C01829=1187.154,242.876,-63.394,-177.309,7.032,148.525
C01830=1187.149,243.125,-63.420,-177.307,7.034,148.524
C01831=1187.146,243.373,-63.446,-177.304,7.037,148.524
C01832=1187.141,243.622,-63.473,-177.302,7.039,148.524
C01833=1187.137,243.871,-63.499,-177.299,7.042,148.524
C01834=1187.132,244.119,-63.526,-177.296,7.044,148.524
C01835=1187.128,244.368,-63.552,-177.293,7.046,148.524
C01836=1187.123,244.616,-63.579,-177.291,7.048,148.523
C01837=1187.119,244.865,-63.605,-177.288,7.050,148.523
C01838=1187.114,245.114,-63.632,-177.286,7.053,148.523
C01839=1187.110,245.361,-63.658,-177.284,7.055,148.523
C01840=1187.105,245.610,-63.684,-177.280,7.058,148.523
C01841=1187.101,245.859,-63.711,-177.278,7.060,148.523
C01842=1187.096,246.107,-63.738,-177.275,7.063,148.522
C01843=1187.091,246.355,-63.765,-177.273,7.065,148.522
C01844=1187.087,246.604,-63.791,-177.270,7.068,148.522
C01845=1187.083,246.853,-63.818,-177.267,7.070,148.522
C01846=1187.079,247.101,-63.844,-177.265,7.073,148.522
C01847=1187.074,247.349,-63.871,-177.262,7.075,148.521
C01848=1187.070,247.599,-63.898,-177.260,7.077,148.521
C01849=1187.066,247.847,-63.924,-177.257,7.080,148.521
C01850=1187.061,248.096,-63.952,-177.255,7.082,148.521
C01851=1187.056,248.344,-63.979,-177.252,7.085,148.521
C01852=1187.053,248.593,-64.005,-177.250,7.087,148.521
C01853=1187.048,248.842,-64.031,-177.246,7.089,148.521
C01854=1187.043,249.090,-64.058,-177.244,7.092,148.520
C01855=1187.039,249.338,-64.085,-177.241,7.094,148.520
C01856=1187.034,249.587,-64.112,-177.239,7.096,148.520
C01857=1187.030,249.835,-64.139,-177.236,7.099,148.520
C01858=1187.026,250.084,-64.165,-177.234,7.101,148.520
C01859=1187.021,250.332,-64.193,-177.231,7.104,148.520
C01860=1187.016,250.581,-64.220,-177.229,7.106,148.520
C01861=1187.012,250.829,-64.247,-177.225,7.109,148.519
C01862=1187.008,251.078,-64.272,-177.223,7.111,148.519
C01863=1187.003,251.326,-64.299,-177.221,7.114,148.519
C01864=1186.999,251.576,-64.327,-177.218,7.116,148.519
C01865=1186.994,251.824,-64.354,-177.215,7.119,148.519
C01866=1186.990,252.072,-64.380,-177.213,7.121,148.519
C01867=1186.986,252.321,-64.408,-177.210,7.124,148.518
C01868=1186.981,252.569,-64.435,-177.208,7.126,148.518
C01869=1186.976,252.818,-64.462,-177.205,7.129,148.518
C01870=1186.972,253.066,-64.488,-177.202,7.131,148.518
C01871=1186.968,253.314,-64.516,-177.200,7.134,148.518
C01872=1186.964,253.563,-64.543,-177.197,7.136,148.518
C01873=1186.959,253.812,-64.570,-177.194,7.139,148.517
C01874=1186.955,254.060,-64.597,-177.192,7.141,148.517
C01875=1186.950,254.309,-64.624,-177.189,7.144,148.517
C01876=1186.946,254.557,-64.651,-177.187,7.146,148.517
C01877=1186.941,254.805,-64.678,-177.184,7.149,148.517
C01878=1186.937,255.054,-64.705,-177.182,7.151,148.517
C01879=1186.933,255.303,-64.733,-177.179,7.153,148.517
C01880=1186.928,255.551,-64.760,-177.176,7.155,148.517
C01881=1186.924,255.799,-64.787,-177.174,7.158,148.516
C01882=1186.919,256.048,-64.814,-177.171,7.160,148.516
C01883=1186.914,256.296,-64.841,-177.168,7.163,148.516
C01884=1186.910,256.545,-64.869,-177.166,7.165,148.516
C01885=1186.907,256.793,-64.896,-177.163,7.168,148.516
C01886=1186.902,257.042,-64.923,-177.161,7.170,148.516
C01887=1186.897,257.290,-64.950,-177.158,7.173,148.516
C01888=1186.893,257.539,-64.977,-177.155,7.176,148.516
C01889=1186.889,257.787,-65.005,-177.153,7.178,148.515
C01890=1186.884,258.036,-65.032,-177.150,7.181,148.515
C01891=1186.880,258.284,-65.060,-177.148,7.183,148.515
C01892=1186.875,258.532,-65.087,-177.145,7.186,148.515
C01893=1186.871,258.781,-65.115,-177.142,7.188,148.515
C01894=1186.867,259.030,-65.142,-177.140,7.191,148.515
C01895=1186.862,259.278,-65.170,-177.138,7.193,148.515
C01896=1186.858,259.526,-65.197,-177.134,7.196,148.514
C01897=1186.854,259.775,-65.224,-177.132,7.198,148.514
C01898=1186.849,260.023,-65.252,-177.129,7.201,148.514
C01899=1186.845,260.272,-65.279,-177.127,7.204,148.514
C01900=1186.840,260.519,-65.307,-177.124,7.206,148.514
C01901=1186.836,260.769,-65.334,-177.121,7.209,148.514
C01902=1186.831,261.017,-65.361,-177.119,7.211,148.514
C01903=1186.827,261.265,-65.389,-177.116,7.214,148.514
C01904=1186.823,261.514,-65.416,-177.114,7.216,148.513
C01905=1186.818,261.762,-65.445,-177.111,7.219,148.513
C01906=1186.813,262.011,-65.472,-177.109,7.221,148.513
C01907=1186.809,262.284,-65.502,-177.106,7.224,148.513
C01908=1186.804,262.557,-65.532,-177.103,7.227,148.513
C01909=1186.799,262.830,-65.563,-177.100,7.230,148.513
C01910=1186.794,263.103,-65.593,-177.097,7.232,148.513
C01911=1186.790,263.350,-65.621,-177.094,7.235,148.513
C01912=1186.786,263.600,-65.648,-177.092,7.237,148.512
C01913=1186.781,263.847,-65.676,-177.089,7.240,148.512
C01914=1186.777,264.097,-65.704,-177.087,7.243,148.512
C01915=1186.772,264.345,-65.732,-177.084,7.245,148.512
C01916=1186.768,264.593,-65.760,-177.081,7.248,148.512
C01917=1186.764,264.842,-65.787,-177.079,7.250,148.512
C01918=1186.760,265.090,-65.815,-177.077,7.253,148.512
C01919=1186.755,265.338,-65.843,-177.074,7.255,148.512
C01920=1186.750,265.587,-65.871,-177.071,7.258,148.511
C01921=1186.746,265.835,-65.899,-177.068,7.261,148.511
C01922=1186.742,266.083,-65.926,-177.066,7.263,148.511
C01923=1186.738,266.332,-65.954,-177.064,7.266,148.511
C01924=1186.733,266.580,-65.981,-177.061,7.268,148.511
C01925=1186.729,266.829,-66.010,-177.058,7.271,148.511
C01926=1186.724,267.077,-66.038,-177.055,7.274,148.511
C01927=1186.720,267.325,-66.065,-177.053,7.276,148.511
C01928=1186.715,267.574,-66.094,-177.051,7.279,148.511
C01929=1186.711,267.822,-66.122,-177.048,7.281,148.511
C01930=1186.707,268.071,-66.150,-177.045,7.284,148.510
C01931=1186.703,268.319,-66.177,-177.042,7.287,148.510
C01932=1186.698,268.568,-66.206,-177.040,7.289,148.510
C01933=1186.694,268.816,-66.233,-177.038,7.292,148.510
C01934=1186.689,269.064,-66.261,-177.035,7.295,148.510
C01935=1186.685,269.313,-66.290,-177.032,7.297,148.510
C01936=1186.681,269.560,-66.318,-177.030,7.300,148.510
C01937=1186.676,269.810,-66.345,-177.027,7.302,148.510
C01938=1186.671,270.058,-66.373,-177.025,7.305,148.510
C01939=1186.668,270.306,-66.402,-177.022,7.308,148.510
C01940=1186.663,270.554,-66.429,-177.020,7.310,148.510
C01941=1186.659,270.803,-66.458,-177.017,7.313,148.509
C01942=1186.654,271.051,-66.486,-177.014,7.315,148.509
C01943=1186.650,271.300,-66.515,-177.012,7.318,148.509
C01944=1186.646,271.548,-66.542,-177.009,7.321,148.509
C01945=1186.642,271.796,-66.570,-177.007,7.323,148.509
C01946=1186.637,272.045,-66.599,-177.004,7.326,148.509
C01947=1186.633,272.293,-66.627,-177.001,7.329,148.509
C01948=1186.628,272.541,-66.655,-176.999,7.331,148.509
C01949=1186.624,272.790,-66.684,-176.996,7.334,148.509
C01950=1186.619,273.038,-66.712,-176.993,7.337,148.509
C01951=1186.615,273.287,-66.740,-176.991,7.339,148.509
C01952=1186.610,273.535,-66.768,-176.988,7.342,148.509
C01953=1186.607,273.783,-66.797,-176.986,7.345,148.508
C01954=1186.601,274.032,-66.825,-176.984,7.347,148.508
C01955=1186.598,274.280,-66.853,-176.981,7.350,148.508
C01956=1186.594,274.528,-66.882,-176.978,7.352,148.508
C01957=1186.589,274.776,-66.910,-176.975,7.355,148.508
C01958=1186.585,275.025,-66.939,-176.973,7.358,148.508
C01959=1186.580,275.273,-66.967,-176.971,7.360,148.508
C01960=1186.576,275.522,-66.996,-176.968,7.363,148.508
C01961=1186.571,275.770,-67.023,-176.965,7.366,148.508
C01962=1186.567,276.018,-67.053,-176.963,7.369,148.508
C01963=1186.564,276.267,-67.081,-176.960,7.372,148.508
C01964=1186.558,276.515,-67.109,-176.958,7.375,148.508
C01965=1186.555,276.764,-67.137,-176.955,7.376,148.507
C01966=1186.550,277.012,-67.166,-176.952,7.379,148.507
C01967=1186.545,277.260,-67.195,-176.949,7.382,148.507
C01968=1186.542,277.509,-67.223,-176.947,7.385,148.507
C01969=1186.537,277.757,-67.252,-176.945,7.388,148.507
C01970=1186.533,278.005,-67.281,-176.942,7.391,148.507
C01971=1186.529,278.254,-67.309,-176.940,7.393,148.507
C01972=1186.524,278.502,-67.338,-176.937,7.396,148.507
C01973=1186.520,278.750,-67.367,-176.934,7.399,148.507
C01974=1186.515,278.998,-67.395,-176.932,7.401,148.507
C01975=1186.511,279.246,-67.423,-176.929,7.404,148.507
C01976=1186.507,279.495,-67.453,-176.926,7.406,148.507
C01977=1186.502,279.743,-67.481,-176.923,7.409,148.507
C01978=1186.498,279.992,-67.509,-176.921,7.412,148.507
C01979=1186.494,280.240,-67.539,-176.919,7.415,148.506
C01980=1186.489,280.488,-67.567,-176.916,7.418,148.506
C01981=1186.485,280.736,-67.596,-176.914,7.420,148.506
C01982=1186.481,280.985,-67.625,-176.911,7.423,148.506
C01983=1186.477,281.233,-67.654,-176.908,7.426,148.506
C01984=1186.472,281.481,-67.682,-176.906,7.428,148.506
C01985=1186.468,281.730,-67.710,-176.903,7.431,148.506
C01986=1186.464,281.978,-67.740,-176.901,7.434,148.506
C01987=1186.459,282.226,-67.768,-176.899,7.436,148.506
C01988=1186.455,282.475,-67.798,-176.896,7.439,148.506
C01989=1186.450,282.723,-67.827,-176.893,7.442,148.506
C01990=1186.447,282.971,-67.855,-176.890,7.445,148.506
C01991=1186.442,283.219,-67.884,-176.888,7.447,148.506
C01992=1186.437,283.468,-67.913,-176.885,7.450,148.506
C01993=1186.433,283.716,-67.943,-176.883,7.453,148.506
C01994=1186.428,283.964,-67.971,-176.881,7.455,148.506
C01995=1186.425,284.212,-68.000,-176.878,7.458,148.506
C01996=1186.421,284.461,-68.029,-176.875,7.461,148.506
C01997=1186.416,284.709,-68.058,-176.872,7.464,148.506
C01998=1186.411,284.957,-68.087,-176.870,7.467,148.506
C01999=1186.407,285.205,-68.117,-176.867,7.469,148.505
C02000=1186.403,285.454,-68.145,-176.864,7.472,148.505
C02001=1186.399,285.702,-68.174,-176.862,7.474,148.505
C02002=1186.395,285.950,-68.204,-176.860,7.477,148.505
C02003=1186.390,286.199,-68.232,-176.857,7.480,148.505
C02004=1186.386,286.447,-68.261,-176.854,7.483,148.505
C02005=1186.381,286.695,-68.291,-176.852,7.486,148.505
C02006=1186.377,286.943,-68.320,-176.849,7.489,148.505
C02007=1186.373,287.192,-68.349,-176.846,7.492,148.505
C02008=1186.368,287.440,-68.378,-176.844,7.495,148.505
C02009=1186.364,287.688,-68.408,-176.842,7.497,148.505
C02010=1186.360,287.936,-68.437,-176.839,7.500,148.505
C02011=1186.355,288.211,-68.469,-176.836,7.503,148.505
C02012=1186.350,288.486,-68.501,-176.833,7.506,148.505
C02013=1186.345,288.760,-68.534,-176.831,7.509,148.505
C02014=1186.340,289.035,-68.566,-176.827,7.513,148.505
C02015=1186.336,289.283,-68.596,-176.825,7.515,148.505
C02016=1186.332,289.532,-68.625,-176.823,7.518,148.505
C02017=1186.327,289.779,-68.654,-176.820,7.521,148.505
C02018=1186.323,290.028,-68.684,-176.818,7.523,148.505
C02019=1186.319,290.276,-68.713,-176.815,7.526,148.505
C02020=1186.315,290.524,-68.743,-176.812,7.529,148.505
C02021=1186.311,290.772,-68.772,-176.810,7.532,148.504
C02022=1186.306,291.021,-68.802,-176.807,7.534,148.504
C02023=1186.302,291.269,-68.831,-176.805,7.537,148.504
C02024=1186.298,291.517,-68.860,-176.802,7.540,148.504
C02025=1186.293,291.765,-68.890,-176.800,7.543,148.505
C02026=1186.289,292.013,-68.919,-176.798,7.545,148.504
C02027=1186.285,292.261,-68.948,-176.795,7.548,148.504
C02028=1186.281,292.510,-68.978,-176.792,7.551,148.504
C02029=1186.277,292.758,-69.007,-176.789,7.554,148.504
C02030=1186.272,293.006,-69.037,-176.787,7.557,148.504
C02031=1186.268,293.254,-69.066,-176.785,7.560,148.504
C02032=1186.263,293.503,-69.096,-176.782,7.563,148.504
C02033=1186.259,293.751,-69.126,-176.779,7.566,148.504
C02034=1186.255,293.999,-69.155,-176.776,7.569,148.504
C02035=1186.251,294.248,-69.185,-176.774,7.571,148.504
C02036=1186.247,294.496,-69.214,-176.771,7.574,148.504
C02037=1186.243,294.744,-69.244,-176.769,7.577,148.504
C02038=1186.238,294.992,-69.274,-176.766,7.580,148.504
C02039=1186.234,295.240,-69.304,-176.764,7.582,148.504
C02040=1186.229,295.489,-69.333,-176.762,7.585,148.504
C02041=1186.225,295.737,-69.363,-176.759,7.588,148.504
C02042=1186.221,295.985,-69.392,-176.756,7.591,148.504
C02043=1186.217,296.233,-69.422,-176.754,7.594,148.504
C02044=1186.212,296.482,-69.452,-176.751,7.596,148.504
C02045=1186.208,296.730,-69.482,-176.749,7.599,148.504
C02046=1186.204,296.978,-69.511,-176.746,7.602,148.504
C02047=1186.200,297.226,-69.541,-176.743,7.605,148.504
C02048=1186.195,297.474,-69.572,-176.741,7.608,148.504
C02049=1186.191,297.723,-69.601,-176.739,7.611,148.504
C02050=1186.187,297.970,-69.631,-176.736,7.614,148.504
C02051=1186.182,298.219,-69.661,-176.733,7.617,148.504
C02052=1186.178,298.467,-69.691,-176.731,7.620,148.504
C02053=1186.174,298.715,-69.721,-176.728,7.622,148.504
C02054=1186.170,298.963,-69.750,-176.726,7.625,148.504
C02055=1186.165,299.212,-69.780,-176.723,7.628,148.504
C02056=1186.161,299.459,-69.810,-176.720,7.631,148.504
C02057=1186.157,299.707,-69.840,-176.718,7.634,148.504
C02058=1186.152,299.955,-69.871,-176.716,7.637,148.504
C02059=1186.148,300.204,-69.900,-176.713,7.640,148.504
C02060=1186.144,300.451,-69.930,-176.711,7.643,148.504
C02061=1186.139,300.700,-69.960,-176.708,7.646,148.504
C02062=1186.136,300.948,-69.991,-176.705,7.649,148.504
C02063=1186.131,301.197,-70.021,-176.703,7.651,148.504
C02064=1186.127,301.444,-70.051,-176.701,7.654,148.504
C02065=1186.123,301.693,-70.081,-176.698,7.657,148.504
C02066=1186.118,301.941,-70.111,-176.695,7.660,148.504
C02067=1186.114,302.189,-70.141,-176.693,7.663,148.504
C02068=1186.110,302.437,-70.172,-176.690,7.665,148.504
C02069=1186.105,302.685,-70.201,-176.688,7.668,148.504
C02070=1186.101,302.933,-70.232,-176.685,7.672,148.504
C02071=1186.097,303.182,-70.262,-176.683,7.675,148.504
C02072=1186.093,303.430,-70.292,-176.680,7.678,148.504
C02073=1186.089,303.678,-70.323,-176.678,7.680,148.504
C02074=1186.085,303.926,-70.352,-176.675,7.683,148.504
C02075=1186.080,304.174,-70.383,-176.672,7.686,148.504
C02076=1186.076,304.422,-70.412,-176.670,7.689,148.504
C02077=1186.071,304.670,-70.443,-176.667,7.692,148.504
C02078=1186.067,304.919,-70.474,-176.665,7.695,148.504
C02079=1186.063,305.166,-70.504,-176.663,7.697,148.504
C02080=1186.058,305.415,-70.534,-176.660,7.700,148.504
C02081=1186.055,305.663,-70.564,-176.658,7.704,148.504
C02082=1186.050,305.911,-70.595,-176.655,7.707,148.504
C02083=1186.046,306.159,-70.625,-176.652,7.710,148.504
C02084=1186.042,306.408,-70.656,-176.649,7.713,148.504
C02085=1186.038,306.655,-70.686,-176.647,7.715,148.504
C02086=1186.033,306.903,-70.717,-176.645,7.718,148.504
C02087=1186.029,307.151,-70.748,-176.642,7.721,148.504
C02088=1186.024,307.399,-70.777,-176.640,7.724,148.504
C02089=1186.020,307.648,-70.808,-176.637,7.727,148.504
C02090=1186.017,307.896,-70.838,-176.635,7.730,148.504
C02091=1186.012,308.144,-70.869,-176.633,7.733,148.504
C02092=1186.007,308.392,-70.900,-176.630,7.736,148.504
C02093=1186.004,308.640,-70.930,-176.627,7.739,148.504
C02094=1185.999,308.889,-70.960,-176.625,7.742,148.505
C02095=1185.994,309.137,-70.991,-176.622,7.745,148.505
C02096=1185.991,309.384,-71.021,-176.619,7.748,148.505
C02097=1185.987,309.633,-71.052,-176.617,7.750,148.504
C02098=1185.982,309.881,-71.083,-176.615,7.753,148.505
C02099=1185.978,310.128,-71.113,-176.612,7.756,148.505
C02100=1185.974,310.376,-71.144,-176.610,7.759,148.505
C02101=1185.969,310.625,-71.175,-176.607,7.762,148.505
C02102=1185.966,310.873,-71.205,-176.605,7.766,148.505
C02103=1185.961,311.121,-71.236,-176.602,7.768,148.505
C02104=1185.957,311.369,-71.267,-176.600,7.771,148.505
C02105=1185.952,311.617,-71.298,-176.598,7.774,148.505
C02106=1185.949,311.865,-71.328,-176.595,7.777,148.505
C02107=1185.944,312.113,-71.359,-176.592,7.780,148.505
C02108=1185.940,312.362,-71.390,-176.589,7.783,148.505
C02109=1185.935,312.609,-71.421,-176.587,7.786,148.505
C02110=1185.931,312.857,-71.451,-176.585,7.789,148.505
C02111=1185.928,313.105,-71.483,-176.582,7.792,148.505
C02112=1185.923,313.353,-71.514,-176.580,7.795,148.505
C02113=1185.918,313.601,-71.544,-176.577,7.798,148.505
C02114=1185.914,313.850,-71.576,-176.575,7.801,148.505
C02115=1185.910,314.126,-71.610,-176.572,7.804,148.505
C02116=1185.905,314.403,-71.644,-176.570,7.807,148.505
C02117=1185.900,314.679,-71.679,-176.566,7.811,148.505
C02118=1185.895,314.955,-71.713,-176.564,7.814,148.505
C02119=1185.891,315.204,-71.744,-176.561,7.817,148.506
C02120=1185.887,315.452,-71.775,-176.559,7.820,148.506
C02121=1185.884,315.700,-71.806,-176.556,7.823,148.506
C02122=1185.879,315.948,-71.837,-176.554,7.827,148.506
C02123=1185.875,316.196,-71.868,-176.552,7.829,148.506
C02124=1185.871,316.444,-71.899,-176.549,7.832,148.506
C02125=1185.866,316.692,-71.930,-176.547,7.835,148.506
C02126=1185.862,316.940,-71.962,-176.544,7.838,148.506
C02127=1185.858,317.188,-71.992,-176.541,7.841,148.506
C02128=1185.853,317.436,-72.023,-176.539,7.845,148.506
C02129=1185.849,317.684,-72.055,-176.536,7.848,148.506
C02130=1185.845,317.932,-72.086,-176.534,7.850,148.506
C02131=1185.841,318.181,-72.117,-176.532,7.853,148.506
C02132=1185.837,318.428,-72.148,-176.529,7.856,148.506
C02133=1185.833,318.676,-72.179,-176.527,7.859,148.506
C02134=1185.829,318.924,-72.210,-176.524,7.862,148.506
C02135=1185.825,319.172,-72.242,-176.521,7.865,148.506
C02136=1185.821,319.420,-72.273,-176.519,7.869,148.507
C02137=1185.817,319.668,-72.304,-176.516,7.872,148.507
C02138=1185.812,319.916,-72.335,-176.514,7.875,148.507
C02139=1185.808,320.164,-72.366,-176.512,7.877,148.507
C02140=1185.804,320.412,-72.398,-176.509,7.880,148.507
C02141=1185.799,320.660,-72.429,-176.507,7.884,148.507
C02142=1185.795,320.908,-72.460,-176.504,7.887,148.507
C02143=1185.790,321.156,-72.492,-176.502,7.890,148.507
C02144=1185.787,321.404,-72.524,-176.499,7.893,148.507
C02145=1185.782,321.652,-72.555,-176.497,7.896,148.507
C02146=1185.778,321.900,-72.587,-176.494,7.899,148.507
C02147=1185.774,322.149,-72.618,-176.493,7.902,148.508
C02148=1185.770,322.396,-72.649,-176.490,7.905,148.508
C02149=1185.766,322.645,-72.680,-176.487,7.908,148.508
C02150=1185.762,322.892,-72.712,-176.485,7.911,148.508
C02151=1185.758,323.140,-72.744,-176.482,7.914,148.508
C02152=1185.753,323.388,-72.775,-176.480,7.917,148.508
C02153=1185.750,323.636,-72.806,-176.477,7.920,148.508
C02154=1185.745,323.884,-72.838,-176.475,7.924,148.508
C02155=1185.741,324.132,-72.870,-176.472,7.927,148.508
C02156=1185.736,324.380,-72.901,-176.470,7.930,148.508
C02157=1185.732,324.628,-72.933,-176.468,7.932,148.508
C02158=1185.729,324.876,-72.965,-176.466,7.935,148.509
C02159=1185.724,325.124,-72.996,-176.463,7.938,148.509
C02160=1185.720,325.372,-73.027,-176.461,7.942,148.509
C02161=1185.715,325.619,-73.059,-176.458,7.945,148.509
C02162=1185.712,325.868,-73.091,-176.456,7.948,148.509
C02163=1185.708,326.116,-73.122,-176.453,7.951,148.509
C02164=1185.703,326.364,-73.154,-176.451,7.954,148.509
C02165=1185.699,326.612,-73.186,-176.448,7.957,148.509
C02166=1185.695,326.859,-73.218,-176.446,7.961,148.509
C02167=1185.691,327.107,-73.250,-176.444,7.963,148.509
C02168=1185.687,327.355,-73.282,-176.442,7.966,148.509
C02169=1185.682,327.604,-73.313,-176.439,7.969,148.509
C02170=1185.678,327.852,-73.345,-176.437,7.973,148.510
C02171=1185.674,328.099,-73.376,-176.434,7.976,148.510
C02172=1185.670,328.347,-73.408,-176.432,7.979,148.510
C02173=1185.666,328.595,-73.441,-176.429,7.982,148.510
C02174=1185.661,328.843,-73.472,-176.427,7.985,148.510
C02175=1185.658,329.091,-73.504,-176.424,7.989,148.510
C02176=1185.653,329.339,-73.536,-176.422,7.992,148.510
C02177=1185.649,329.586,-73.568,-176.419,7.995,148.511
C02178=1185.645,329.834,-73.600,-176.418,7.997,148.511
C02179=1185.641,330.083,-73.632,-176.415,8.000,148.511
C02180=1185.636,330.330,-73.664,-176.413,8.004,148.511
C02181=1185.633,330.578,-73.695,-176.410,8.007,148.511
C02182=1185.628,330.827,-73.728,-176.408,8.010,148.511
C02183=1185.624,331.074,-73.759,-176.406,8.013,148.511
C02184=1185.620,331.322,-73.792,-176.403,8.016,148.511
C02185=1185.616,331.570,-73.824,-176.401,8.020,148.512
C02186=1185.612,331.818,-73.855,-176.398,8.023,148.512
C02187=1185.607,332.066,-73.887,-176.396,8.026,148.512
C02188=1185.603,332.314,-73.919,-176.393,8.029,148.512
C02189=1185.599,332.562,-73.952,-176.391,8.032,148.512
C02190=1185.595,332.809,-73.984,-176.389,8.035,148.512
C02191=1185.591,333.057,-74.016,-176.387,8.038,148.512
C02192=1185.587,333.305,-74.048,-176.384,8.041,148.512
C02193=1185.583,333.553,-74.080,-176.382,8.044,148.513
C02194=1185.578,333.801,-74.112,-176.380,8.048,148.513
C02195=1185.574,334.049,-74.144,-176.377,8.051,148.513
C02196=1185.570,334.297,-74.177,-176.375,8.054,148.513
C02197=1185.567,334.545,-74.209,-176.372,8.057,148.513
C02198=1185.561,334.793,-74.241,-176.370,8.061,148.513
C02199=1185.558,335.041,-74.273,-176.367,8.064,148.513
C02200=1185.554,335.288,-74.306,-176.365,8.067,148.514
C02201=1185.550,335.536,-74.338,-176.363,8.070,148.514
C02202=1185.545,335.785,-74.370,-176.360,8.073,148.514
C02203=1185.541,336.032,-74.403,-176.358,8.077,148.514
C02204=1185.537,336.280,-74.435,-176.356,8.079,148.514
C02205=1185.533,336.528,-74.467,-176.354,8.083,148.514
C02206=1185.529,336.776,-74.500,-176.351,8.086,148.514
C02207=1185.525,337.024,-74.532,-176.349,8.089,148.515
C02208=1185.520,337.271,-74.564,-176.347,8.092,148.515
C02209=1185.516,337.519,-74.597,-176.344,8.095,148.515
C02210=1185.512,337.767,-74.630,-176.342,8.098,148.515
C02211=1185.508,338.015,-74.662,-176.340,8.102,148.515
C02212=1185.504,338.263,-74.695,-176.337,8.105,148.515
C02213=1185.500,338.510,-74.726,-176.335,8.108,148.516
C02214=1185.496,338.758,-74.759,-176.333,8.112,148.516
C02215=1185.491,339.006,-74.792,-176.330,8.115,148.516
C02216=1185.488,339.254,-74.824,-176.328,8.118,148.516
C02217=1185.483,339.502,-74.857,-176.326,8.121,148.516
C02218=1185.479,339.750,-74.890,-176.323,8.125,148.517
C02219=1185.475,340.029,-74.926,-176.321,8.128,148.517
C02220=1185.470,340.308,-74.962,-176.318,8.131,148.517
C02221=1185.465,340.587,-74.999,-176.316,8.135,148.517
C02222=1185.460,340.865,-75.036,-176.313,8.139,148.517
C02223=1185.456,341.113,-75.069,-176.311,8.142,148.518
C02224=1185.452,341.361,-75.101,-176.309,8.145,148.518
C02225=1185.448,341.609,-75.134,-176.307,8.148,148.518
C02226=1185.444,341.857,-75.167,-176.304,8.152,148.518
C02227=1185.440,342.105,-75.200,-176.302,8.155,148.518
C02228=1185.436,342.352,-75.232,-176.299,8.158,148.518
C02229=1185.432,342.601,-75.265,-176.297,8.161,148.519
C02230=1185.428,342.848,-75.298,-176.295,8.165,148.519
C02231=1185.423,343.095,-75.331,-176.293,8.168,148.519
C02232=1185.419,343.343,-75.362,-176.290,8.171,148.519
C02233=1185.415,343.591,-75.396,-176.288,8.175,148.519
C02234=1185.411,343.839,-75.429,-176.286,8.178,148.520
C02235=1185.407,344.087,-75.461,-176.284,8.181,148.520
C02236=1185.402,344.335,-75.494,-176.281,8.185,148.520
C02237=1185.398,344.583,-75.528,-176.279,8.188,148.520
C02238=1185.395,344.830,-75.560,-176.277,8.191,148.521
C02239=1185.390,345.078,-75.593,-176.275,8.195,148.521
C02240=1185.386,345.326,-75.626,-176.273,8.197,148.521
C02241=1185.382,345.574,-75.659,-176.271,8.200,148.521
C02242=1185.378,345.822,-75.692,-176.268,8.204,148.521
C02243=1185.374,346.069,-75.725,-176.266,8.207,148.522
C02244=1185.370,346.317,-75.758,-176.264,8.210,148.522
C02245=1185.366,346.565,-75.790,-176.262,8.214,148.522
C02246=1185.362,346.813,-75.823,-176.259,8.217,148.522
C02247=1185.358,347.060,-75.856,-176.257,8.220,148.522
C02248=1185.354,347.308,-75.890,-176.255,8.224,148.523
C02249=1185.349,347.556,-75.923,-176.253,8.227,148.523
C02250=1185.345,347.804,-75.956,-176.250,8.230,148.523
C02251=1185.341,348.051,-75.989,-176.248,8.234,148.523
C02252=1185.337,348.299,-76.022,-176.246,8.237,148.524
C02253=1185.333,348.547,-76.055,-176.244,8.240,148.524
C02254=1185.329,348.795,-76.089,-176.241,8.244,148.524
C02255=1185.325,349.042,-76.122,-176.239,8.247,148.524
C02256=1185.321,349.290,-76.155,-176.237,8.250,148.524
C02257=1185.316,349.538,-76.188,-176.235,8.254,148.525
C02258=1185.312,349.785,-76.221,-176.233,8.257,148.525
C02259=1185.308,350.033,-76.254,-176.230,8.260,148.525
C02260=1185.304,350.281,-76.287,-176.228,8.264,148.526
C02261=1185.300,350.529,-76.321,-176.226,8.267,148.526
C02262=1185.296,350.776,-76.354,-176.224,8.270,148.526
C02263=1185.292,351.025,-76.387,-176.221,8.274,148.526
C02264=1185.288,351.273,-76.420,-176.220,8.277,148.527
C02265=1185.284,351.520,-76.454,-176.217,8.281,148.527
C02266=1185.280,351.768,-76.487,-176.215,8.284,148.527
C02267=1185.276,352.016,-76.520,-176.213,8.287,148.527
C02268=1185.272,352.263,-76.554,-176.211,8.291,148.528
C02269=1185.268,352.511,-76.587,-176.209,8.294,148.528
C02270=1185.263,352.758,-76.620,-176.207,8.297,148.528
C02271=1185.259,353.006,-76.654,-176.205,8.300,148.528
C02272=1185.254,353.254,-76.687,-176.203,8.303,148.529
C02273=1185.251,353.503,-76.721,-176.201,8.307,148.529
C02274=1185.247,353.750,-76.754,-176.199,8.310,148.529
C02275=1185.243,353.997,-76.788,-176.196,8.314,148.529
C02276=1185.239,354.245,-76.821,-176.194,8.317,148.530
C02277=1185.235,354.493,-76.854,-176.192,8.321,148.530
C02278=1185.231,354.740,-76.888,-176.190,8.324,148.530
C02279=1185.226,354.988,-76.922,-176.188,8.327,148.531
C02280=1185.222,355.236,-76.955,-176.186,8.331,148.531
C02281=1185.219,355.484,-76.989,-176.184,8.334,148.531
C02282=1185.214,355.731,-77.022,-176.181,8.337,148.531
C02283=1185.210,355.979,-77.055,-176.180,8.341,148.532
C02284=1185.207,356.226,-77.089,-176.177,8.344,148.532
C02285=1185.202,356.475,-77.123,-176.176,8.348,148.532
C02286=1185.198,356.723,-77.156,-176.173,8.351,148.533
C02287=1185.194,356.970,-77.190,-176.171,8.355,148.533
C02288=1185.190,357.217,-77.223,-176.169,8.358,148.533
C02289=1185.186,357.465,-77.258,-176.167,8.362,148.534
C02290=1185.182,357.713,-77.291,-176.165,8.365,148.534
C02291=1185.178,357.961,-77.325,-176.163,8.369,148.534
C02292=1185.174,358.208,-77.358,-176.161,8.372,148.534
C02293=1185.169,358.456,-77.392,-176.159,8.376,148.535
C02294=1185.165,358.703,-77.426,-176.157,8.379,148.535
C02295=1185.162,358.952,-77.460,-176.155,8.382,148.536
C02296=1185.158,359.199,-77.493,-176.152,8.386,148.536
C02297=1185.153,359.447,-77.527,-176.151,8.389,148.536
C02298=1185.149,359.694,-77.561,-176.148,8.393,148.536
C02299=1185.146,359.942,-77.595,-176.147,8.396,148.537
C02300=1185.141,360.190,-77.629,-176.145,8.400,148.537
C02301=1185.137,360.437,-77.663,-176.143,8.403,148.538
C02302=1185.134,360.685,-77.696,-176.141,8.407,148.538
C02303=1185.129,360.933,-77.731,-176.139,8.409,148.538
C02304=1185.125,361.180,-77.764,-176.137,8.413,148.539
C02305=1185.121,361.428,-77.798,-176.135,8.417,148.539
C02306=1185.117,361.676,-77.833,-176.133,8.420,148.539
C02307=1185.113,361.923,-77.866,-176.131,8.424,148.540
C02308=1185.109,362.171,-77.900,-176.130,8.427,148.540
C02309=1185.105,362.419,-77.934,-176.127,8.431,148.540
C02310=1185.101,362.666,-77.968,-176.126,8.434,148.541
C02311=1185.097,362.914,-78.002,-176.124,8.438,148.541
C02312=1185.093,363.162,-78.036,-176.122,8.441,148.542
C02313=1185.089,363.409,-78.070,-176.120,8.444,148.542
C02314=1185.085,363.657,-78.104,-176.118,8.448,148.542
C02315=1185.081,363.905,-78.138,-176.117,8.451,148.543
C02316=1185.077,364.153,-78.172,-176.115,8.455,148.543
C02317=1185.073,364.400,-78.206,-176.113,8.458,148.544
C02318=1185.069,364.648,-78.241,-176.111,8.462,148.544
C02319=1185.065,364.895,-78.275,-176.109,8.465,148.544
C02320=1185.061,365.142,-78.309,-176.108,8.468,148.545
C02321=1185.057,365.391,-78.343,-176.106,8.472,148.545
C02322=1185.053,365.638,-78.377,-176.104,8.475,148.545
C02323=1185.048,365.920,-78.416,-176.102,8.479,148.546
C02324=1185.044,366.201,-78.455,-176.100,8.483,148.546
C02325=1185.039,366.481,-78.493,-176.098,8.487,148.547
C02326=1185.034,366.763,-78.533,-176.097,8.491,148.547
C02327=1185.031,367.012,-78.566,-176.095,8.495,148.548
C02328=1185.026,367.259,-78.601,-176.093,8.498,148.548
C02329=1185.022,367.506,-78.635,-176.092,8.501,148.549
C02330=1185.018,367.754,-78.669,-176.090,8.505,148.549
C02331=1185.014,368.002,-78.704,-176.088,8.508,148.550
C02332=1185.010,368.249,-78.738,-176.086,8.512,148.550
C02333=1185.006,368.497,-78.773,-176.085,8.515,148.550
C02334=1185.002,368.744,-78.807,-176.083,8.518,148.551
C02335=1184.998,368.992,-78.841,-176.081,8.522,148.551
C02336=1184.994,369.239,-78.875,-176.080,8.526,148.552
C02337=1184.991,369.487,-78.910,-176.079,8.529,148.552
C02338=1184.986,369.735,-78.945,-176.077,8.532,148.553
C02339=1184.982,369.982,-78.978,-176.075,8.536,148.553
C02340=1184.978,370.230,-79.013,-176.074,8.539,148.553
C02341=1184.974,370.477,-79.047,-176.072,8.542,148.554
C02342=1184.970,370.725,-79.082,-176.071,8.546,148.555
C02343=1184.966,370.973,-79.116,-176.070,8.549,148.555
C02344=1184.963,371.220,-79.151,-176.068,8.553,148.555
C02345=1184.958,371.468,-79.185,-176.066,8.557,148.556
C02346=1184.954,371.716,-79.220,-176.065,8.559,148.556
C02347=1184.950,371.963,-79.254,-176.063,8.563,148.557
C02348=1184.946,372.210,-79.288,-176.063,8.566,148.557
C02349=1184.942,372.458,-79.324,-176.061,8.570,148.558
C02350=1184.938,372.705,-79.358,-176.059,8.573,148.558
C02351=1184.934,372.953,-79.393,-176.058,8.576,148.559
C02352=1184.930,373.201,-79.427,-176.056,8.580,148.559
C02353=1184.926,373.448,-79.461,-176.055,8.583,148.560
C02354=1184.922,373.696,-79.496,-176.054,8.587,148.560
C02355=1184.918,373.943,-79.531,-176.052,8.590,148.561
C02356=1184.914,374.191,-79.566,-176.051,8.594,148.561
C02357=1184.910,374.439,-79.600,-176.050,8.596,148.562
C02358=1184.906,374.686,-79.634,-176.048,8.600,148.562
C02359=1184.902,374.934,-79.669,-176.047,8.603,148.563
C02360=1184.897,375.181,-79.704,-176.046,8.607,148.563
C02361=1184.894,375.429,-79.739,-176.045,8.610,148.564
C02362=1184.890,375.676,-79.773,-176.043,8.614,148.564
C02363=1184.886,375.924,-79.808,-176.042,8.617,148.565
C02364=1184.881,376.171,-79.843,-176.041,8.620,148.565
C02365=1184.878,376.419,-79.877,-176.040,8.623,148.566
C02366=1184.874,376.667,-79.912,-176.039,8.627,148.567
C02367=1184.870,376.914,-79.947,-176.037,8.630,148.567
C02368=1184.866,377.162,-79.982,-176.036,8.633,148.568
C02369=1184.861,377.409,-80.017,-176.035,8.636,148.568
C02370=1184.859,377.657,-80.052,-176.034,8.640,148.569
C02371=1184.854,377.904,-80.086,-176.033,8.643,148.569
C02372=1184.850,378.152,-80.121,-176.032,8.646,148.570
C02373=1184.846,378.399,-80.156,-176.030,8.650,148.570
C02374=1184.842,378.647,-80.191,-176.029,8.653,148.571
C02375=1184.837,378.894,-80.225,-176.029,8.656,148.571
C02376=1184.834,379.142,-80.260,-176.027,8.660,148.572
C02377=1184.830,379.390,-80.295,-176.026,8.663,148.572
C02378=1184.826,379.637,-80.330,-176.025,8.666,148.573
C02379=1184.822,379.885,-80.365,-176.024,8.669,148.574
C02380=1184.817,380.132,-80.400,-176.023,8.673,148.574
C02381=1184.814,380.380,-80.435,-176.022,8.676,148.575
C02382=1184.809,380.627,-80.470,-176.021,8.679,148.575
C02383=1184.806,380.874,-80.505,-176.021,8.682,148.576
C02384=1184.802,381.122,-80.539,-176.019,8.685,148.576
C02385=1184.798,381.369,-80.575,-176.018,8.689,148.577
C02386=1184.794,381.617,-80.609,-176.017,8.692,148.578
C02387=1184.790,381.864,-80.645,-176.016,8.695,148.578
C02388=1184.786,382.112,-80.680,-176.015,8.698,148.579
C02389=1184.782,382.360,-80.715,-176.015,8.701,148.579
C02390=1184.778,382.607,-80.750,-176.014,8.704,148.580
C02391=1184.774,382.855,-80.785,-176.013,8.707,148.580
C02392=1184.769,383.102,-80.820,-176.012,8.711,148.581
C02393=1184.766,383.349,-80.855,-176.011,8.714,148.582
C02394=1184.762,383.598,-80.890,-176.011,8.717,148.582
C02395=1184.758,383.844,-80.925,-176.010,8.720,148.583
C02396=1184.754,384.093,-80.960,-176.009,8.723,148.583
C02397=1184.751,384.340,-80.995,-176.008,8.726,148.584
C02398=1184.746,384.586,-81.030,-176.007,8.729,148.585
C02399=1184.742,384.835,-81.065,-176.007,8.733,148.585
C02400=1184.739,385.082,-81.100,-176.006,8.736,148.586
C02401=1184.734,385.330,-81.135,-176.005,8.739,148.587
C02402=1184.731,385.577,-81.170,-176.005,8.742,148.587
C02403=1184.726,385.824,-81.206,-176.004,8.745,148.588
C02404=1184.722,386.072,-81.240,-176.003,8.747,148.588
C02405=1184.719,386.319,-81.276,-176.003,8.750,148.589
C02406=1184.714,386.567,-81.310,-176.002,8.754,148.590
C02407=1184.710,386.814,-81.346,-176.001,8.757,148.590
C02408=1184.707,387.062,-81.382,-176.001,8.760,148.591
C02409=1184.702,387.309,-81.416,-176.000,8.762,148.591
C02410=1184.699,387.557,-81.452,-176.000,8.765,148.592
C02411=1184.695,387.804,-81.487,-175.999,8.769,148.593
C02412=1184.690,388.052,-81.522,-175.998,8.772,148.593
C02413=1184.687,388.299,-81.557,-175.998,8.774,148.594
C02414=1184.683,388.547,-81.593,-175.997,8.777,148.594
C02415=1184.679,388.794,-81.628,-175.997,8.780,148.595
C02416=1184.674,389.042,-81.663,-175.997,8.783,148.596
C02417=1184.670,389.289,-81.699,-175.996,8.786,148.596
C02418=1184.667,389.537,-81.734,-175.996,8.789,148.597
C02419=1184.662,389.784,-81.769,-175.995,8.791,148.598
C02420=1184.658,390.032,-81.804,-175.994,8.795,148.598
C02421=1184.655,390.279,-81.840,-175.994,8.797,148.599
C02422=1184.650,390.526,-81.875,-175.994,8.800,148.599
C02423=1184.647,390.774,-81.910,-175.994,8.802,148.600
C02424=1184.643,391.022,-81.946,-175.993,8.806,148.600
C02425=1184.639,391.269,-81.981,-175.993,8.808,148.601
C02426=1184.635,391.516,-82.016,-175.992,8.811,148.602
C02427=1184.630,391.800,-82.056,-175.992,8.815,148.603
C02428=1184.626,392.084,-82.097,-175.991,8.818,148.603
C02429=1184.622,392.368,-82.138,-175.991,8.820,148.604
C02430=1184.617,392.652,-82.179,-175.991,8.824,148.605
C02431=1184.613,392.899,-82.214,-175.990,8.827,148.605
C02432=1184.608,393.147,-82.249,-175.990,8.829,148.606
C02433=1184.605,393.394,-82.284,-175.990,8.832,148.607
C02434=1184.601,393.642,-82.320,-175.989,8.835,148.607
C02435=1184.597,393.889,-82.356,-175.989,8.837,148.608
C02436=1184.593,394.136,-82.391,-175.989,8.840,148.608
C02437=1184.589,394.384,-82.426,-175.989,8.843,148.609
C02438=1184.586,394.631,-82.462,-175.988,8.845,148.610
C02439=1184.581,394.880,-82.497,-175.989,8.848,148.610
C02440=1184.577,395.126,-82.532,-175.988,8.851,148.611
C02441=1184.573,395.374,-82.568,-175.987,8.853,148.611
C02442=1184.569,395.621,-82.604,-175.988,8.856,148.612
C02443=1184.566,395.869,-82.639,-175.987,8.858,148.613
C02444=1184.561,396.116,-82.674,-175.987,8.861,148.614
C02445=1184.557,396.363,-82.710,-175.987,8.864,148.614
C02446=1184.553,396.611,-82.746,-175.987,8.866,148.615
C02447=1184.549,396.858,-82.780,-175.987,8.868,148.615
C02448=1184.545,397.106,-82.816,-175.986,8.872,148.616
C02449=1184.542,397.353,-82.852,-175.986,8.874,148.617
C02450=1184.538,397.601,-82.887,-175.986,8.876,148.617
C02451=1184.533,397.849,-82.923,-175.986,8.879,148.618
C02452=1184.529,398.095,-82.958,-175.986,8.881,148.618
C02453=1184.526,398.343,-82.994,-175.985,8.884,148.619
C02454=1184.522,398.590,-83.030,-175.986,8.886,148.620
C02455=1184.518,398.838,-83.065,-175.985,8.889,148.620
C02456=1184.513,399.085,-83.101,-175.985,8.892,148.621
C02457=1184.510,399.333,-83.136,-175.985,8.894,148.621
C02458=1184.506,399.580,-83.172,-175.984,8.896,148.622
C02459=1184.502,399.828,-83.207,-175.985,8.899,148.623
C02460=1184.498,400.074,-83.243,-175.984,8.901,148.623
C02461=1184.494,400.322,-83.279,-175.985,8.904,148.624
C02462=1184.490,400.570,-83.314,-175.984,8.906,148.624
C02463=1184.486,400.817,-83.350,-175.984,8.908,148.625
C02464=1184.483,401.065,-83.385,-175.984,8.911,148.626
C02465=1184.478,401.311,-83.421,-175.984,8.913,148.626
C02466=1184.474,401.559,-83.457,-175.984,8.916,148.627
C02467=1184.470,401.807,-83.492,-175.984,8.918,148.627
C02468=1184.467,402.054,-83.528,-175.984,8.920,148.628
C02469=1184.462,402.301,-83.563,-175.984,8.923,148.629
C02470=1184.458,402.549,-83.599,-175.984,8.925,148.629
C02471=1184.454,402.796,-83.635,-175.983,8.927,148.630
C02472=1184.451,403.044,-83.670,-175.984,8.930,148.630
C02473=1184.447,403.291,-83.706,-175.983,8.932,148.631
C02474=1184.442,403.539,-83.742,-175.983,8.935,148.632
C02475=1184.438,403.786,-83.777,-175.984,8.936,148.632
C02476=1184.435,404.034,-83.813,-175.983,8.938,148.633
C02477=1184.431,404.281,-83.848,-175.984,8.941,148.633
C02478=1184.427,404.529,-83.884,-175.983,8.943,148.634
C02479=1184.422,404.776,-83.920,-175.983,8.945,148.634
C02480=1184.419,405.023,-83.955,-175.983,8.948,148.635
C02481=1184.415,405.271,-83.991,-175.983,8.950,148.636
C02482=1184.411,405.518,-84.027,-175.983,8.952,148.636
C02483=1184.407,405.766,-84.062,-175.984,8.954,148.637
C02484=1184.403,406.013,-84.098,-175.983,8.957,148.637
C02485=1184.399,406.260,-84.133,-175.983,8.959,148.638
C02486=1184.395,406.508,-84.169,-175.983,8.961,148.639
C02487=1184.391,406.755,-84.205,-175.983,8.964,148.639
C02488=1184.388,407.002,-84.241,-175.983,8.965,148.640
C02489=1184.384,407.250,-84.277,-175.983,8.967,148.640
C02490=1184.379,407.497,-84.312,-175.983,8.970,148.641
C02491=1184.375,407.745,-84.348,-175.983,8.972,148.641
C02492=1184.372,407.992,-84.383,-175.983,8.974,148.642
C02493=1184.367,408.240,-84.420,-175.983,8.976,148.643
C02494=1184.363,408.487,-84.455,-175.983,8.978,148.643
C02495=1184.360,408.735,-84.491,-175.983,8.981,148.644
C02496=1184.356,408.982,-84.526,-175.983,8.982,148.644
C02497=1184.351,409.229,-84.563,-175.983,8.985,148.645
C02498=1184.348,409.476,-84.598,-175.983,8.987,148.645
C02499=1184.344,409.724,-84.634,-175.983,8.989,148.646
C02500=1184.340,409.972,-84.670,-175.983,8.991,148.646
C02501=1184.336,410.219,-84.706,-175.983,8.993,148.647
C02502=1184.332,410.467,-84.741,-175.983,8.995,148.648
C02503=1184.327,410.714,-84.777,-175.983,8.997,148.648
C02504=1184.324,410.961,-84.813,-175.983,8.999,148.649
C02505=1184.320,411.208,-84.849,-175.983,9.001,148.649
C02506=1184.316,411.456,-84.885,-175.984,9.003,148.650
C02507=1184.312,411.703,-84.920,-175.983,9.005,148.650
C02508=1184.309,411.951,-84.956,-175.983,9.008,148.651
C02509=1184.304,412.198,-84.992,-175.983,9.009,148.651
C02510=1184.300,412.445,-85.028,-175.983,9.011,148.652
C02511=1184.297,412.692,-85.063,-175.983,9.014,148.652
C02512=1184.292,412.940,-85.100,-175.984,9.015,148.653
C02513=1184.289,413.188,-85.135,-175.983,9.018,148.653
C02514=1184.285,413.435,-85.171,-175.984,9.019,148.654
C02515=1184.281,413.682,-85.208,-175.983,9.021,148.654
C02516=1184.277,413.929,-85.243,-175.983,9.024,148.655
C02517=1184.273,414.177,-85.278,-175.983,9.025,148.655
C02518=1184.268,414.425,-85.314,-175.984,9.028,148.656
C02519=1184.265,414.672,-85.350,-175.984,9.029,148.657
C02520=1184.261,414.919,-85.386,-175.984,9.031,148.657
C02521=1184.257,415.167,-85.422,-175.983,9.034,148.658
C02522=1184.253,415.414,-85.458,-175.984,9.035,148.658
C02523=1184.250,415.629,-85.489,-175.983,9.037,148.659
C02524=1184.246,415.844,-85.520,-175.984,9.039,148.659
C02525=1184.244,416.059,-85.551,-175.984,9.040,148.659
C02526=1184.243,416.274,-85.582,-175.983,9.042,148.660
C02527=1184.242,416.489,-85.613,-175.984,9.044,148.660
C02528=1184.242,416.703,-85.644,-175.983,9.045,148.661
C02529=1184.244,416.918,-85.675,-175.984,9.046,148.661
C02530=1184.246,417.132,-85.706,-175.983,9.048,148.662
C02531=1183.825,417.132,-85.747,-175.986,9.059,148.665
C02532=1183.822,416.917,-85.716,-175.987,9.057,148.665
C02533=1183.821,416.701,-85.685,-175.987,9.056,148.664
C02534=1183.821,416.485,-85.655,-175.987,9.054,148.664
C02535=1183.821,416.269,-85.623,-175.986,9.053,148.663
C02536=1183.822,416.052,-85.592,-175.987,9.051,148.663
C02537=1183.825,415.836,-85.561,-175.987,9.049,148.663
C02538=1183.829,415.619,-85.530,-175.986,9.048,148.662
C02539=1183.832,415.403,-85.498,-175.987,9.046,148.662
C02540=1183.836,415.155,-85.462,-175.986,9.044,148.661
C02541=1183.840,414.908,-85.426,-175.987,9.042,148.661
C02542=1183.843,414.661,-85.390,-175.987,9.040,148.660
C02543=1183.848,414.414,-85.354,-175.987,9.038,148.660
C02544=1183.852,414.166,-85.319,-175.987,9.036,148.659
C02545=1183.855,413.919,-85.283,-175.987,9.035,148.659
C02546=1183.860,413.671,-85.247,-175.986,9.032,148.658
C02547=1183.863,413.424,-85.211,-175.986,9.031,148.658
C02548=1183.867,413.176,-85.175,-175.986,9.028,148.657
C02549=1183.871,412.929,-85.139,-175.987,9.026,148.657
C02550=1183.876,412.682,-85.104,-175.986,9.025,148.656
C02551=1183.879,412.434,-85.068,-175.987,9.022,148.656
C02552=1183.883,412.187,-85.032,-175.986,9.020,148.655
C02553=1183.887,411.940,-84.996,-175.986,9.018,148.654
C02554=1183.891,411.692,-84.960,-175.986,9.016,148.654
C02555=1183.895,411.444,-84.924,-175.987,9.014,148.653
C02556=1183.899,411.197,-84.889,-175.986,9.012,148.653
C02557=1183.903,410.951,-84.853,-175.986,9.010,148.652
C02558=1183.907,410.703,-84.817,-175.986,9.008,148.652
C02559=1183.911,410.455,-84.781,-175.986,9.006,148.651
C02560=1183.914,410.208,-84.746,-175.986,9.004,148.651
C02561=1183.919,409.960,-84.709,-175.986,9.001,148.650
C02562=1183.922,409.713,-84.674,-175.986,9.000,148.649
C02563=1183.926,409.465,-84.638,-175.986,8.998,148.649
C02564=1183.931,409.219,-84.602,-175.986,8.995,148.648
C02565=1183.934,408.971,-84.566,-175.986,8.994,148.648
C02566=1183.938,408.724,-84.531,-175.986,8.991,148.647
C02567=1183.942,408.476,-84.495,-175.986,8.989,148.647
C02568=1183.946,408.228,-84.459,-175.986,8.987,148.646
C02569=1183.950,407.981,-84.424,-175.986,8.985,148.646
C02570=1183.954,407.734,-84.388,-175.986,8.983,148.645
C02571=1183.958,407.487,-84.351,-175.986,8.981,148.645
C02572=1183.962,407.239,-84.316,-175.986,8.978,148.644
C02573=1183.966,406.992,-84.280,-175.986,8.977,148.643
C02574=1183.970,406.744,-84.244,-175.986,8.974,148.643
C02575=1183.974,406.496,-84.209,-175.986,8.972,148.642
C02576=1183.978,406.250,-84.174,-175.986,8.969,148.642
C02577=1183.981,406.002,-84.138,-175.986,8.968,148.641
C02578=1183.986,405.754,-84.102,-175.986,8.966,148.641
C02579=1183.990,405.507,-84.066,-175.986,8.963,148.640
C02580=1183.993,405.259,-84.031,-175.986,8.961,148.639
C02581=1183.997,405.013,-83.996,-175.986,8.958,148.639
C02582=1184.002,404.765,-83.959,-175.986,8.956,148.638
C02583=1184.005,404.518,-83.923,-175.986,8.955,148.638
C02584=1184.009,404.270,-83.888,-175.986,8.952,148.637
C02585=1184.013,404.023,-83.851,-175.986,8.950,148.636
C02586=1184.017,403.775,-83.816,-175.986,8.948,148.636
C02587=1184.021,403.528,-83.781,-175.986,8.945,148.635
C02588=1184.025,403.281,-83.745,-175.986,8.943,148.635
C02589=1184.029,403.033,-83.709,-175.987,8.940,148.634
C02590=1184.033,402.785,-83.673,-175.986,8.938,148.633
C02591=1184.037,402.538,-83.638,-175.987,8.936,148.633
C02592=1184.041,402.291,-83.603,-175.986,8.933,148.632
C02593=1184.045,402.043,-83.567,-175.987,8.931,148.632
C02594=1184.049,401.796,-83.531,-175.987,8.929,148.631
C02595=1184.053,401.548,-83.496,-175.987,8.926,148.630
C02596=1184.056,401.301,-83.460,-175.986,8.925,148.630
C02597=1184.061,401.054,-83.425,-175.986,8.922,148.629
C02598=1184.065,400.806,-83.389,-175.987,8.920,148.629
C02599=1184.069,400.559,-83.353,-175.987,8.917,148.628
C02600=1184.072,400.311,-83.318,-175.987,8.914,148.627
C02601=1184.077,400.064,-83.282,-175.987,8.912,148.627
C02602=1184.081,399.817,-83.246,-175.987,8.909,148.626
C02603=1184.085,399.569,-83.211,-175.988,8.907,148.626
C02604=1184.088,399.322,-83.175,-175.987,8.904,148.625
C02605=1184.092,399.074,-83.140,-175.988,8.902,148.624
C02606=1184.096,398.827,-83.104,-175.988,8.900,148.624
C02607=1184.101,398.579,-83.068,-175.988,8.897,148.623
C02608=1184.104,398.332,-83.033,-175.988,8.895,148.623
C02609=1184.108,398.084,-82.997,-175.988,8.892,148.622
C02610=1184.112,397.838,-82.962,-175.988,8.890,148.621
C02611=1184.116,397.590,-82.926,-175.988,8.887,148.621
C02612=1184.120,397.342,-82.890,-175.989,8.885,148.620
C02613=1184.124,397.094,-82.855,-175.989,8.882,148.620
C02614=1184.128,396.847,-82.820,-175.989,8.880,148.619
C02615=1184.132,396.600,-82.785,-175.989,8.877,148.618
C02616=1184.136,396.352,-82.749,-175.989,8.875,148.618
C02617=1184.139,396.105,-82.714,-175.990,8.872,148.617
C02618=1184.144,395.858,-82.678,-175.989,8.869,148.616
C02619=1184.148,395.610,-82.642,-175.990,8.867,148.616
C02620=1184.152,395.363,-82.607,-175.990,8.865,148.615
C02621=1184.155,395.115,-82.571,-175.990,8.861,148.614
C02622=1184.160,394.869,-82.536,-175.991,8.859,148.614
C02623=1184.164,394.620,-82.501,-175.990,8.856,148.613
C02624=1184.167,394.373,-82.466,-175.991,8.853,148.613
C02625=1184.172,394.125,-82.430,-175.991,8.851,148.612
C02626=1184.176,393.878,-82.394,-175.991,8.848,148.611
C02627=1184.180,393.631,-82.359,-175.992,8.845,148.611
C02628=1184.183,393.383,-82.323,-175.992,8.843,148.610
C02629=1184.187,393.136,-82.288,-175.992,8.841,148.609
C02630=1184.192,392.888,-82.253,-175.993,8.837,148.609
C02631=1184.195,392.641,-82.218,-175.993,8.835,148.608
C02632=1184.200,392.358,-82.177,-175.993,8.832,148.607
C02633=1184.205,392.073,-82.136,-175.994,8.828,148.607
C02634=1184.209,391.789,-82.095,-175.994,8.825,148.606
C02635=1184.214,391.505,-82.055,-175.994,8.822,148.605
C02636=1184.217,391.258,-82.019,-175.995,8.819,148.605
C02637=1184.222,391.011,-81.984,-175.995,8.817,148.604
C02638=1184.225,390.763,-81.949,-175.996,8.814,148.603
C02639=1184.229,390.515,-81.914,-175.996,8.811,148.603
C02640=1184.233,390.268,-81.879,-175.996,8.808,148.602
C02641=1184.237,390.021,-81.843,-175.997,8.805,148.602
C02642=1184.241,389.773,-81.808,-175.997,8.803,148.601
C02643=1184.245,389.525,-81.773,-175.998,8.799,148.600
C02644=1184.249,389.278,-81.738,-175.998,8.797,148.600
C02645=1184.253,389.031,-81.702,-175.999,8.794,148.599
C02646=1184.257,388.783,-81.666,-176.000,8.791,148.599
C02647=1184.262,388.536,-81.631,-175.999,8.788,148.598
C02648=1184.265,388.288,-81.596,-176.000,8.785,148.597
C02649=1184.269,388.041,-81.560,-176.001,8.782,148.597
C02650=1184.274,387.793,-81.526,-176.001,8.779,148.596
C02651=1184.277,387.546,-81.490,-176.002,8.776,148.595
C02652=1184.281,387.298,-81.455,-176.003,8.773,148.595
C02653=1184.285,387.052,-81.420,-176.003,8.770,148.594
C02654=1184.289,386.803,-81.385,-176.003,8.768,148.593
C02655=1184.293,386.556,-81.349,-176.004,8.765,148.593
C02656=1184.297,386.309,-81.314,-176.005,8.761,148.592
C02657=1184.301,386.061,-81.279,-176.006,8.758,148.592
C02658=1184.305,385.813,-81.244,-176.006,8.755,148.591
C02659=1184.309,385.566,-81.209,-176.007,8.752,148.591
C02660=1184.313,385.319,-81.174,-176.007,8.750,148.590
C02661=1184.317,385.071,-81.138,-176.008,8.747,148.589
C02662=1184.321,384.824,-81.104,-176.009,8.743,148.589
C02663=1184.325,384.576,-81.068,-176.009,8.740,148.588
C02664=1184.328,384.329,-81.033,-176.010,8.737,148.587
C02665=1184.333,384.081,-80.998,-176.011,8.734,148.587
C02666=1184.337,383.834,-80.963,-176.012,8.731,148.586
C02667=1184.341,383.586,-80.928,-176.013,8.728,148.586
C02668=1184.345,383.339,-80.893,-176.014,8.725,148.585
C02669=1184.348,383.091,-80.858,-176.014,8.722,148.585
C02670=1184.352,382.844,-80.823,-176.015,8.719,148.584
C02671=1184.356,382.596,-80.788,-176.016,8.716,148.583
C02672=1184.360,382.349,-80.753,-176.017,8.712,148.583
C02673=1184.365,382.101,-80.718,-176.018,8.709,148.582
C02674=1184.368,381.854,-80.683,-176.018,8.706,148.582
C02675=1184.372,381.606,-80.648,-176.020,8.702,148.581
C02676=1184.377,381.359,-80.613,-176.021,8.699,148.580
C02677=1184.380,381.111,-80.578,-176.021,8.696,148.580
C02678=1184.385,380.864,-80.543,-176.022,8.693,148.579
C02679=1184.389,380.616,-80.508,-176.023,8.690,148.579
C02680=1184.393,380.369,-80.473,-176.024,8.687,148.578
C02681=1184.396,380.121,-80.438,-176.025,8.683,148.577
C02682=1184.400,379.874,-80.403,-176.027,8.680,148.577
C02683=1184.404,379.626,-80.368,-176.027,8.677,148.577
C02684=1184.408,379.379,-80.333,-176.028,8.674,148.576
C02685=1184.413,379.131,-80.298,-176.029,8.670,148.575
C02686=1184.417,378.883,-80.264,-176.030,8.667,148.575
C02687=1184.420,378.636,-80.228,-176.031,8.664,148.574
C02688=1184.425,378.388,-80.194,-176.033,8.660,148.574
C02689=1184.428,378.141,-80.159,-176.034,8.657,148.573
C02690=1184.432,377.894,-80.124,-176.035,8.654,148.573
C02691=1184.436,377.645,-80.089,-176.036,8.650,148.572
C02692=1184.441,377.399,-80.054,-176.037,8.647,148.572
C02693=1184.445,377.151,-80.019,-176.038,8.644,148.571
C02694=1184.448,376.903,-79.985,-176.039,8.640,148.570
C02695=1184.452,376.656,-79.950,-176.041,8.638,148.570
C02696=1184.457,376.409,-79.915,-176.042,8.634,148.569
C02697=1184.461,376.160,-79.881,-176.043,8.631,148.569
C02698=1184.464,375.913,-79.845,-176.044,8.628,148.568
C02699=1184.468,375.666,-79.811,-176.045,8.624,148.568
C02700=1184.472,375.418,-79.776,-176.047,8.621,148.567
C02701=1184.477,375.170,-79.742,-176.048,8.617,148.567
C02702=1184.480,374.923,-79.706,-176.049,8.614,148.566
C02703=1184.484,374.676,-79.672,-176.051,8.610,148.566
C02704=1184.488,374.428,-79.638,-176.052,8.608,148.565
C02705=1184.493,374.180,-79.603,-176.053,8.604,148.565
C02706=1184.497,373.932,-79.568,-176.055,8.601,148.564
C02707=1184.500,373.686,-79.534,-176.056,8.597,148.564
C02708=1184.504,373.437,-79.499,-176.057,8.594,148.563
C02709=1184.509,373.190,-79.464,-176.059,8.590,148.563
C02710=1184.512,372.942,-79.430,-176.060,8.587,148.562
C02711=1184.517,372.695,-79.396,-176.061,8.583,148.562
C02712=1184.520,372.447,-79.360,-176.063,8.580,148.561
C02713=1184.525,372.200,-79.326,-176.064,8.577,148.561
C02714=1184.528,371.952,-79.291,-176.066,8.573,148.560
C02715=1184.533,371.705,-79.257,-176.067,8.570,148.560
C02716=1184.537,371.457,-79.223,-176.069,8.567,148.559
C02717=1184.540,371.209,-79.188,-176.070,8.563,148.559
C02718=1184.545,370.962,-79.154,-176.071,8.560,148.558
C02719=1184.549,370.714,-79.119,-176.073,8.556,148.558
C02720=1184.553,370.467,-79.085,-176.075,8.553,148.557
C02721=1184.557,370.219,-79.050,-176.076,8.550,148.557
C02722=1184.561,369.971,-79.016,-176.078,8.546,148.556
C02723=1184.564,369.723,-78.982,-176.079,8.542,148.556
C02724=1184.569,369.476,-78.947,-176.081,8.540,148.556
C02725=1184.573,369.229,-78.913,-176.082,8.536,148.555
C02726=1184.577,368.981,-78.878,-176.084,8.532,148.555
C02727=1184.581,368.734,-78.845,-176.086,8.528,148.554
C02728=1184.585,368.485,-78.810,-176.087,8.526,148.554
C02729=1184.589,368.238,-78.775,-176.089,8.522,148.553
C02730=1184.592,367.990,-78.741,-176.090,8.518,148.553
C02731=1184.597,367.743,-78.707,-176.092,8.515,148.552
C02732=1184.601,367.496,-78.673,-176.094,8.512,148.552
C02733=1184.605,367.248,-78.638,-176.095,8.508,148.552
C02734=1184.609,367.000,-78.604,-176.097,8.505,148.551
C02735=1184.613,366.753,-78.570,-176.099,8.501,148.551
C02736=1184.617,366.472,-78.531,-176.100,8.497,148.550
C02737=1184.622,366.190,-78.491,-176.102,8.494,148.550
C02738=1184.627,365.908,-78.453,-176.105,8.489,148.549
C02739=1184.631,365.627,-78.414,-176.106,8.485,148.549
C02740=1184.635,365.379,-78.380,-176.108,8.482,148.548
C02741=1184.639,365.132,-78.345,-176.110,8.478,148.548
C02742=1184.643,364.884,-78.311,-176.111,8.475,148.547
C02743=1184.647,364.636,-78.278,-176.113,8.472,148.547
C02744=1184.651,364.388,-78.243,-176.115,8.469,148.547
C02745=1184.655,364.141,-78.209,-176.117,8.465,148.546
C02746=1184.660,363.894,-78.175,-176.119,8.461,148.546
C02747=1184.663,363.646,-78.140,-176.121,8.458,148.546
C02748=1184.667,363.398,-78.107,-176.123,8.454,148.545
C02749=1184.672,363.151,-78.073,-176.124,8.452,148.545
C02750=1184.675,362.903,-78.039,-176.126,8.448,148.544
C02751=1184.680,362.655,-78.005,-176.128,8.444,148.544
C02752=1184.684,362.408,-77.971,-176.130,8.441,148.544
C02753=1184.687,362.160,-77.937,-176.132,8.437,148.543
C02754=1184.692,361.912,-77.903,-176.134,8.434,148.543
C02755=1184.696,361.665,-77.869,-176.136,8.430,148.543
C02756=1184.700,361.418,-77.835,-176.138,8.427,148.542
C02757=1184.704,361.169,-77.801,-176.140,8.423,148.542
C02758=1184.707,360.922,-77.767,-176.141,8.420,148.541
C02759=1184.712,360.675,-77.733,-176.144,8.416,148.541
C02760=1184.716,360.426,-77.699,-176.145,8.413,148.541
C02761=1184.719,360.179,-77.665,-176.147,8.410,148.541
C02762=1184.724,359.931,-77.632,-176.149,8.406,148.540
C02763=1184.728,359.684,-77.598,-176.151,8.403,148.540
C02764=1184.732,359.435,-77.564,-176.153,8.400,148.540
C02765=1184.736,359.188,-77.530,-176.155,8.396,148.539
C02766=1184.740,358.940,-77.497,-176.157,8.393,148.539
C02767=1184.744,358.693,-77.463,-176.159,8.389,148.538
C02768=1184.748,358.445,-77.429,-176.161,8.386,148.538
C02769=1184.752,358.197,-77.395,-176.163,8.382,148.538
C02770=1184.756,357.950,-77.362,-176.165,8.379,148.538
C02771=1184.760,357.703,-77.328,-176.167,8.375,148.537
C02772=1184.764,357.454,-77.294,-176.169,8.372,148.537
C02773=1184.768,357.207,-77.260,-176.172,8.368,148.537
C02774=1184.773,356.959,-77.227,-176.173,8.365,148.536
C02775=1184.777,356.711,-77.193,-176.176,8.362,148.536
C02776=1184.780,356.464,-77.160,-176.178,8.358,148.536
C02777=1184.785,356.215,-77.125,-176.180,8.355,148.535
C02778=1184.789,355.968,-77.092,-176.182,8.351,148.535
C02779=1184.793,355.721,-77.058,-176.184,8.348,148.535
C02780=1184.797,355.473,-77.025,-176.186,8.344,148.534
C02781=1184.801,355.226,-76.991,-176.188,8.341,148.534
C02782=1184.806,354.978,-76.958,-176.191,8.338,148.534
C02783=1184.809,354.729,-76.924,-176.192,8.334,148.534
C02784=1184.813,354.481,-76.891,-176.195,8.331,148.533
C02785=1184.817,354.234,-76.857,-176.197,8.327,148.533
C02786=1184.821,353.987,-76.824,-176.199,8.324,148.533
C02787=1184.825,353.739,-76.791,-176.201,8.320,148.532
C02788=1184.829,353.492,-76.757,-176.203,8.317,148.532
C02789=1184.834,353.244,-76.723,-176.205,8.314,148.532
C02790=1184.838,352.995,-76.690,-176.207,8.310,148.532
C02791=1184.842,352.748,-76.656,-176.209,8.307,148.531
C02792=1184.846,352.500,-76.623,-176.212,8.304,148.531
C02793=1184.850,352.252,-76.590,-176.214,8.300,148.531
C02794=1184.854,352.005,-76.556,-176.216,8.297,148.531
C02795=1184.858,351.757,-76.523,-176.218,8.293,148.530
C02796=1184.862,351.510,-76.490,-176.220,8.290,148.530
C02797=1184.866,351.262,-76.457,-176.223,8.287,148.530
C02798=1184.870,351.014,-76.424,-176.225,8.283,148.530
C02799=1184.874,350.766,-76.390,-176.227,8.280,148.529
C02800=1184.878,350.518,-76.357,-176.229,8.276,148.529
C02801=1184.882,350.270,-76.324,-176.231,8.273,148.529
C02802=1184.886,350.022,-76.291,-176.233,8.270,148.529
C02803=1184.890,349.775,-76.258,-176.236,8.266,148.528
C02804=1184.894,349.528,-76.224,-176.238,8.263,148.528
C02805=1184.898,349.280,-76.191,-176.240,8.260,148.528
C02806=1184.903,349.032,-76.157,-176.242,8.256,148.527
C02807=1184.907,348.784,-76.124,-176.244,8.253,148.527
C02808=1184.911,348.537,-76.091,-176.246,8.250,148.527
C02809=1184.915,348.288,-76.059,-176.248,8.247,148.527
C02810=1184.919,348.041,-76.025,-176.250,8.244,148.527
C02811=1184.924,347.793,-75.992,-176.253,8.240,148.526
C02812=1184.928,347.545,-75.959,-176.255,8.237,148.526
C02813=1184.932,347.297,-75.926,-176.257,8.234,148.526
C02814=1184.936,347.050,-75.893,-176.259,8.230,148.526
C02815=1184.940,346.802,-75.860,-176.262,8.227,148.526
C02816=1184.944,346.554,-75.827,-176.264,8.224,148.525
C02817=1184.948,346.307,-75.793,-176.266,8.221,148.525
C02818=1184.953,346.059,-75.760,-176.268,8.217,148.525
C02819=1184.956,345.811,-75.728,-176.271,8.214,148.525
C02820=1184.960,345.563,-75.695,-176.273,8.211,148.524
C02821=1184.965,345.315,-75.662,-176.275,8.207,148.524
C02822=1184.969,345.068,-75.629,-176.277,8.204,148.524
C02823=1184.973,344.820,-75.596,-176.280,8.201,148.524
C02824=1184.977,344.572,-75.563,-176.282,8.197,148.524
C02825=1184.981,344.324,-75.530,-176.284,8.194,148.523
C02826=1184.985,344.076,-75.498,-176.286,8.191,148.523
C02827=1184.989,343.829,-75.464,-176.289,8.187,148.523
C02828=1184.993,343.580,-75.432,-176.291,8.184,148.523
C02829=1184.998,343.333,-75.399,-176.293,8.181,148.522
C02830=1185.002,343.085,-75.366,-176.295,8.177,148.522
C02831=1185.006,342.836,-75.333,-176.298,8.174,148.522
C02832=1185.010,342.589,-75.301,-176.300,8.171,148.522
C02833=1185.014,342.342,-75.268,-176.302,8.167,148.522
C02834=1185.019,342.094,-75.235,-176.305,8.164,148.522
C02835=1185.023,341.846,-75.202,-176.307,8.161,148.521
C02836=1185.026,341.599,-75.170,-176.309,8.158,148.521
C02837=1185.031,341.350,-75.137,-176.311,8.155,148.521
C02838=1185.035,341.102,-75.104,-176.313,8.152,148.521
C02839=1185.039,340.854,-75.072,-176.316,8.149,148.521
C02840=1185.044,340.576,-75.035,-176.318,8.145,148.520
C02841=1185.048,340.297,-74.999,-176.321,8.142,148.520
C02842=1185.053,340.018,-74.961,-176.324,8.137,148.520
C02843=1185.058,339.740,-74.925,-176.326,8.134,148.520
C02844=1185.062,339.491,-74.892,-176.329,8.131,148.520
C02845=1185.066,339.244,-74.860,-176.331,8.127,148.519
C02846=1185.070,338.995,-74.827,-176.333,8.124,148.519
C02847=1185.074,338.748,-74.795,-176.336,8.121,148.519
C02848=1185.078,338.500,-74.762,-176.338,8.118,148.519
C02849=1185.082,338.252,-74.729,-176.340,8.114,148.519
C02850=1185.086,338.005,-74.698,-176.343,8.111,148.519
C02851=1185.091,337.756,-74.665,-176.345,8.108,148.519
C02852=1185.095,337.509,-74.632,-176.347,8.105,148.518
C02853=1185.099,337.260,-74.600,-176.350,8.101,148.518
C02854=1185.103,337.013,-74.567,-176.352,8.098,148.518
C02855=1185.107,336.765,-74.535,-176.354,8.096,148.518
C02856=1185.112,336.517,-74.503,-176.356,8.093,148.518
C02857=1185.115,336.270,-74.471,-176.359,8.089,148.518
C02858=1185.119,336.021,-74.438,-176.361,8.086,148.517
C02859=1185.124,335.773,-74.406,-176.364,8.083,148.517
C02860=1185.127,335.526,-74.373,-176.366,8.080,148.517
C02861=1185.132,335.278,-74.341,-176.368,8.076,148.517
C02862=1185.136,335.030,-74.309,-176.370,8.073,148.517
C02863=1185.140,334.781,-74.277,-176.373,8.070,148.517
C02864=1185.144,334.534,-74.244,-176.375,8.067,148.516
C02865=1185.149,334.286,-74.212,-176.378,8.063,148.516
C02866=1185.153,334.038,-74.180,-176.380,8.060,148.516
C02867=1185.157,333.790,-74.148,-176.383,8.057,148.516
C02868=1185.160,333.543,-74.115,-176.385,8.054,148.516
C02869=1185.166,333.295,-74.083,-176.387,8.051,148.516
C02870=1185.169,333.047,-74.051,-176.390,8.047,148.516
C02871=1185.174,332.799,-74.019,-176.391,8.045,148.515
C02872=1185.177,332.551,-73.987,-176.394,8.042,148.515
C02873=1185.182,332.303,-73.956,-176.396,8.039,148.515
C02874=1185.186,332.055,-73.923,-176.399,8.035,148.515
C02875=1185.190,331.807,-73.891,-176.401,8.032,148.515
C02876=1185.194,331.559,-73.858,-176.404,8.029,148.515
C02877=1185.198,331.312,-73.827,-176.406,8.026,148.515
C02878=1185.202,331.064,-73.795,-176.409,8.023,148.515
C02879=1185.206,330.815,-73.762,-176.411,8.019,148.514
C02880=1185.211,330.568,-73.731,-176.413,8.016,148.514
C02881=1185.215,330.320,-73.699,-176.416,8.013,148.514
C02882=1185.219,330.072,-73.667,-176.418,8.010,148.514
C02883=1185.223,329.824,-73.635,-176.421,8.007,148.514
C02884=1185.228,329.576,-73.603,-176.422,8.004,148.514
C02885=1185.231,329.328,-73.571,-176.425,8.001,148.514
C02886=1185.236,329.081,-73.539,-176.427,7.998,148.514
C02887=1185.240,328.832,-73.507,-176.430,7.995,148.513
C02888=1185.244,328.584,-73.475,-176.432,7.992,148.513
C02889=1185.248,328.337,-73.444,-176.435,7.988,148.513
C02890=1185.253,328.088,-73.411,-176.437,7.985,148.513
C02891=1185.256,327.840,-73.379,-176.440,7.982,148.513
C02892=1185.261,327.592,-73.349,-176.442,7.979,148.513
C02893=1185.265,327.344,-73.317,-176.445,7.976,148.513
C02894=1185.270,327.097,-73.285,-176.447,7.972,148.513
C02895=1185.273,326.849,-73.253,-176.450,7.969,148.513
C02896=1185.277,326.601,-73.221,-176.451,7.967,148.512
C02897=1185.281,326.353,-73.190,-176.454,7.964,148.512
C02898=1185.286,326.105,-73.157,-176.456,7.960,148.512
C02899=1185.290,325.857,-73.126,-176.459,7.957,148.512
C02900=1185.294,325.609,-73.095,-176.461,7.954,148.512
C02901=1185.298,325.361,-73.063,-176.464,7.951,148.512
C02902=1185.302,325.114,-73.031,-176.466,7.948,148.512
C02903=1185.307,324.865,-72.999,-176.469,7.945,148.512
C02904=1185.311,324.617,-72.968,-176.471,7.942,148.512
C02905=1185.315,324.369,-72.936,-176.474,7.939,148.512
C02906=1185.319,324.121,-72.904,-176.476,7.935,148.511
C02907=1185.323,323.873,-72.874,-176.478,7.933,148.511
C02908=1185.327,323.625,-72.842,-176.480,7.930,148.511
C02909=1185.332,323.378,-72.810,-176.483,7.927,148.511
C02910=1185.336,323.129,-72.778,-176.485,7.923,148.511
C02911=1185.340,322.882,-72.747,-176.488,7.920,148.511
C02912=1185.344,322.634,-72.715,-176.490,7.917,148.511
C02913=1185.349,322.386,-72.684,-176.493,7.914,148.511
C02914=1185.352,322.138,-72.653,-176.496,7.911,148.511
C02915=1185.357,321.890,-72.622,-176.498,7.908,148.511
C02916=1185.361,321.642,-72.590,-176.500,7.906,148.511
C02917=1185.365,321.394,-72.559,-176.502,7.902,148.510
C02918=1185.369,321.146,-72.527,-176.505,7.899,148.510
C02919=1185.373,320.898,-72.495,-176.507,7.896,148.510
C02920=1185.377,320.650,-72.465,-176.510,7.893,148.510
C02921=1185.382,320.402,-72.433,-176.513,7.890,148.510
C02922=1185.386,320.154,-72.402,-176.515,7.887,148.510
C02923=1185.390,319.906,-72.371,-176.518,7.884,148.510
C02924=1185.394,319.658,-72.340,-176.520,7.880,148.510
C02925=1185.398,319.410,-72.308,-176.522,7.878,148.510
C02926=1185.402,319.162,-72.277,-176.524,7.875,148.510
C02927=1185.407,318.914,-72.246,-176.527,7.872,148.510
C02928=1185.411,318.666,-72.214,-176.530,7.869,148.510
C02929=1185.415,318.418,-72.184,-176.532,7.865,148.510
C02930=1185.419,318.170,-72.152,-176.535,7.862,148.510
C02931=1185.423,317.922,-72.121,-176.538,7.859,148.510
C02932=1185.427,317.673,-72.090,-176.540,7.856,148.509
C02933=1185.432,317.426,-72.058,-176.543,7.853,148.509
C02934=1185.436,317.178,-72.028,-176.544,7.851,148.509
C02935=1185.440,316.929,-71.996,-176.547,7.848,148.509
C02936=1185.445,316.682,-71.965,-176.550,7.845,148.509
C02937=1185.449,316.433,-71.934,-176.552,7.841,148.509
C02938=1185.453,316.185,-71.903,-176.555,7.838,148.509
C02939=1185.458,315.938,-71.872,-176.557,7.835,148.509
C02940=1185.462,315.689,-71.840,-176.560,7.832,148.509
C02941=1185.466,315.441,-71.810,-176.562,7.829,148.509
C02942=1185.470,315.193,-71.779,-176.564,7.827,148.509
C02943=1185.474,314.945,-71.748,-176.567,7.824,148.509
C02944=1185.478,314.668,-71.714,-176.570,7.820,148.509
C02945=1185.484,314.392,-71.679,-176.573,7.817,148.509
C02946=1185.488,314.116,-71.644,-176.575,7.813,148.508
C02947=1185.493,313.839,-71.610,-176.578,7.810,148.508
C02948=1185.497,313.591,-71.580,-176.580,7.807,148.509
C02949=1185.501,313.343,-71.548,-176.583,7.804,148.509
C02950=1185.505,313.095,-71.517,-176.585,7.801,148.508
C02951=1185.510,312.847,-71.486,-176.588,7.798,148.508
C02952=1185.514,312.599,-71.456,-176.591,7.795,148.508
C02953=1185.518,312.350,-71.425,-176.593,7.792,148.508
C02954=1185.523,312.102,-71.394,-176.596,7.789,148.508
C02955=1185.527,311.854,-71.363,-176.598,7.787,148.508
C02956=1185.530,311.606,-71.333,-176.600,7.783,148.508
C02957=1185.535,311.358,-71.302,-176.603,7.780,148.508
C02958=1185.540,311.110,-71.271,-176.606,7.777,148.508
C02959=1185.544,310.862,-71.240,-176.608,7.774,148.508
C02960=1185.548,310.614,-71.210,-176.610,7.771,148.508
C02961=1185.552,310.366,-71.179,-176.613,7.768,148.508
C02962=1185.556,310.117,-71.148,-176.615,7.766,148.508
C02963=1185.560,309.870,-71.118,-176.618,7.763,148.508
C02964=1185.565,309.622,-71.087,-176.620,7.759,148.508
C02965=1185.569,309.374,-71.056,-176.623,7.756,148.508
C02966=1185.573,309.125,-71.026,-176.626,7.753,148.508
C02967=1185.577,308.877,-70.995,-176.628,7.750,148.508
C02968=1185.582,308.629,-70.964,-176.630,7.748,148.508
C02969=1185.586,308.382,-70.934,-176.633,7.745,148.508
C02970=1185.590,308.133,-70.903,-176.636,7.742,148.508
C02971=1185.595,307.885,-70.873,-176.638,7.739,148.508
C02972=1185.598,307.637,-70.843,-176.641,7.736,148.508
C02973=1185.603,307.389,-70.812,-176.643,7.733,148.508
C02974=1185.608,307.141,-70.781,-176.645,7.730,148.508
C02975=1185.611,306.893,-70.751,-176.648,7.727,148.508
C02976=1185.616,306.644,-70.721,-176.650,7.724,148.507
C02977=1185.620,306.396,-70.690,-176.653,7.721,148.507
C02978=1185.624,306.148,-70.660,-176.656,7.718,148.507
C02979=1185.628,305.901,-70.630,-176.659,7.715,148.507
C02980=1185.632,305.652,-70.598,-176.661,7.713,148.508
C02981=1185.637,305.404,-70.568,-176.663,7.710,148.507
C02982=1185.641,305.156,-70.538,-176.666,7.707,148.507
C02983=1185.646,304.908,-70.507,-176.668,7.704,148.507
C02984=1185.650,304.660,-70.478,-176.671,7.701,148.507
C02985=1185.654,304.412,-70.447,-176.673,7.697,148.507
C02986=1185.658,304.163,-70.417,-176.675,7.695,148.507
C02987=1185.663,303.915,-70.387,-176.678,7.692,148.507
C02988=1185.667,303.667,-70.356,-176.681,7.689,148.507
C02989=1185.671,303.419,-70.326,-176.684,7.686,148.507
C02990=1185.675,303.171,-70.296,-176.686,7.683,148.507
C02991=1185.680,302.923,-70.266,-176.689,7.680,148.507
C02992=1185.684,302.675,-70.236,-176.691,7.678,148.507
C02993=1185.687,302.426,-70.206,-176.693,7.675,148.507
C02994=1185.692,302.178,-70.175,-176.696,7.672,148.507
C02995=1185.696,301.930,-70.145,-176.699,7.669,148.507
C02996=1185.701,301.682,-70.115,-176.702,7.666,148.507
C02997=1185.705,301.434,-70.085,-176.703,7.663,148.507
C02998=1185.710,301.186,-70.054,-176.706,7.660,148.507
C02999=1185.714,300.938,-70.025,-176.709,7.657,148.507
C03000=1185.718,300.690,-69.995,-176.711,7.654,148.507
C03001=1185.723,300.442,-69.965,-176.714,7.651,148.507
C03002=1185.727,300.193,-69.935,-176.716,7.649,148.507
C03003=1185.730,299.945,-69.905,-176.719,7.646,148.507
C03004=1185.735,299.696,-69.875,-176.721,7.643,148.507
C03005=1185.739,299.449,-69.844,-176.724,7.640,148.507
C03006=1185.743,299.200,-69.815,-176.727,7.637,148.507
C03007=1185.748,298.952,-69.784,-176.729,7.635,148.507
C03008=1185.752,298.704,-69.755,-176.732,7.632,148.507
C03009=1185.756,298.456,-69.725,-176.734,7.629,148.507
C03010=1185.761,298.208,-69.695,-176.737,7.625,148.507
C03011=1185.765,297.960,-69.665,-176.739,7.622,148.507
C03012=1185.769,297.711,-69.636,-176.741,7.620,148.507
C03013=1185.774,297.463,-69.605,-176.744,7.617,148.507
C03014=1185.778,297.215,-69.575,-176.747,7.614,148.507
C03015=1185.782,296.967,-69.546,-176.750,7.611,148.507
C03016=1185.786,296.719,-69.517,-176.752,7.608,148.507
C03017=1185.791,296.471,-69.486,-176.754,7.606,148.507
C03018=1185.795,296.222,-69.456,-176.757,7.603,148.507
C03019=1185.799,295.974,-69.427,-176.759,7.600,148.507
C03020=1185.803,295.726,-69.397,-176.762,7.597,148.507
C03021=1185.807,295.478,-69.367,-176.764,7.594,148.507
C03022=1185.812,295.230,-69.337,-176.767,7.591,148.507
C03023=1185.816,294.981,-69.308,-176.770,7.588,148.507
C03024=1185.820,294.733,-69.278,-176.772,7.585,148.507
C03025=1185.825,294.485,-69.249,-176.775,7.582,148.507
C03026=1185.829,294.237,-69.219,-176.777,7.580,148.507
C03027=1185.833,293.989,-69.189,-176.780,7.577,148.507
C03028=1185.838,293.740,-69.159,-176.783,7.574,148.507
C03029=1185.842,293.492,-69.130,-176.785,7.571,148.508
C03030=1185.846,293.244,-69.100,-176.788,7.569,148.508
C03031=1185.850,292.996,-69.071,-176.790,7.566,148.507
C03032=1185.854,292.747,-69.041,-176.793,7.563,148.507
C03033=1185.859,292.499,-69.012,-176.795,7.560,148.507
C03034=1185.863,292.251,-68.983,-176.798,7.557,148.507
C03035=1185.867,292.003,-68.953,-176.800,7.555,148.508
C03036=1185.872,291.755,-68.924,-176.803,7.552,148.508
C03037=1185.876,291.507,-68.894,-176.806,7.549,148.508
C03038=1185.881,291.258,-68.864,-176.808,7.546,148.508
C03039=1185.885,291.010,-68.835,-176.810,7.543,148.508
C03040=1185.889,290.762,-68.805,-176.813,7.540,148.508
C03041=1185.893,290.513,-68.776,-176.816,7.537,148.508
C03042=1185.897,290.265,-68.747,-176.819,7.534,148.508
C03043=1185.902,290.017,-68.717,-176.821,7.532,148.508
C03044=1185.906,289.769,-68.688,-176.824,7.529,148.508
C03045=1185.911,289.521,-68.659,-176.826,7.526,148.508
C03046=1185.915,289.273,-68.629,-176.829,7.523,148.508
C03047=1185.919,289.024,-68.600,-176.831,7.521,148.508
C03048=1185.924,288.750,-68.568,-176.834,7.518,148.508
C03049=1185.929,288.475,-68.535,-176.837,7.514,148.508
C03050=1185.933,288.201,-68.503,-176.840,7.511,148.508
C03051=1185.938,287.926,-68.470,-176.843,7.508,148.508
C03052=1185.942,287.677,-68.441,-176.845,7.505,148.508
C03053=1185.947,287.430,-68.412,-176.847,7.503,148.508
C03054=1185.951,287.182,-68.383,-176.850,7.500,148.508
C03055=1185.955,286.933,-68.354,-176.853,7.497,148.508
C03056=1185.959,286.685,-68.325,-176.856,7.494,148.508
C03057=1185.963,286.436,-68.295,-176.858,7.492,148.508
C03058=1185.968,286.188,-68.266,-176.860,7.489,148.508
C03059=1185.973,285.940,-68.238,-176.863,7.486,148.508
C03060=1185.977,285.692,-68.208,-176.865,7.484,148.508
C03061=1185.981,285.443,-68.179,-176.868,7.481,148.509
C03062=1185.986,285.194,-68.150,-176.871,7.478,148.509
C03063=1185.990,284.947,-68.121,-176.873,7.475,148.509
C03064=1185.994,284.699,-68.092,-176.876,7.473,148.509
C03065=1185.998,284.450,-68.063,-176.878,7.470,148.509
C03066=1186.002,284.202,-68.034,-176.881,7.467,148.509
C03067=1186.007,283.954,-68.005,-176.884,7.464,148.509
C03068=1186.012,283.705,-67.976,-176.886,7.462,148.509
C03069=1186.016,283.457,-67.947,-176.889,7.459,148.509
C03070=1186.020,283.208,-67.918,-176.891,7.456,148.509
C03071=1186.024,282.961,-67.889,-176.894,7.453,148.509
C03072=1186.029,282.712,-67.861,-176.896,7.450,148.509
C03073=1186.033,282.464,-67.831,-176.899,7.447,148.509
C03074=1186.037,282.216,-67.802,-176.901,7.445,148.509
C03075=1186.042,281.968,-67.774,-176.904,7.442,148.509
C03076=1186.046,281.719,-67.744,-176.907,7.439,148.509
C03077=1186.050,281.470,-67.716,-176.909,7.436,148.509
C03078=1186.055,281.223,-67.688,-176.911,7.434,148.509
C03079=1186.059,280.974,-67.658,-176.915,7.431,148.510
C03080=1186.063,280.725,-67.630,-176.917,7.428,148.510
C03081=1186.068,280.478,-67.601,-176.920,7.426,148.510
C03082=1186.072,280.229,-67.573,-176.922,7.423,148.510
C03083=1186.076,279.981,-67.543,-176.925,7.420,148.510
C03084=1186.081,279.733,-67.515,-176.927,7.418,148.510
C03085=1186.085,279.484,-67.487,-176.930,7.415,148.510
C03086=1186.089,279.236,-67.457,-176.933,7.412,148.510
C03087=1186.094,278.988,-67.429,-176.935,7.409,148.510
C03088=1186.098,278.740,-67.400,-176.937,7.407,148.510
C03089=1186.102,278.491,-67.371,-176.940,7.404,148.510
C03090=1186.107,278.243,-67.343,-176.943,7.401,148.510
C03091=1186.111,277.995,-67.314,-176.945,7.399,148.510
C03092=1186.115,277.746,-67.285,-176.948,7.396,148.510
C03093=1186.119,277.498,-67.257,-176.951,7.393,148.510
C03094=1186.124,277.249,-67.229,-176.953,7.391,148.511
C03095=1186.128,277.001,-67.199,-176.956,7.388,148.511
C03096=1186.132,276.753,-67.171,-176.959,7.385,148.511
C03097=1186.137,276.504,-67.143,-176.961,7.383,148.511
C03098=1186.141,276.256,-67.115,-176.963,7.380,148.511
C03099=1186.145,276.008,-67.085,-176.966,7.377,148.511
C03100=1186.149,275.759,-67.057,-176.968,7.375,148.511
C03101=1186.154,275.511,-67.029,-176.971,7.372,148.511
C03102=1186.159,275.262,-67.000,-176.974,7.369,148.511
C03103=1186.163,275.014,-66.972,-176.976,7.367,148.511
C03104=1186.168,274.766,-66.944,-176.979,7.364,148.511
C03105=1186.172,274.518,-66.915,-176.982,7.361,148.511
C03106=1186.176,274.269,-66.886,-176.984,7.359,148.511
C03107=1186.180,274.021,-66.858,-176.987,7.356,148.511
C03108=1186.185,273.773,-66.830,-176.989,7.353,148.511
C03109=1186.189,273.524,-66.802,-176.992,7.351,148.512
C03110=1186.193,273.276,-66.774,-176.994,7.348,148.512
C03111=1186.198,273.027,-66.745,-176.997,7.345,148.512
C03112=1186.202,272.779,-66.717,-177.000,7.343,148.512
C03113=1186.206,272.531,-66.689,-177.002,7.340,148.512
C03114=1186.211,272.283,-66.661,-177.005,7.338,148.512
C03115=1186.215,272.034,-66.632,-177.007,7.335,148.512
C03116=1186.220,271.786,-66.604,-177.010,7.332,148.512
C03117=1186.224,271.537,-66.576,-177.012,7.329,148.512
C03118=1186.228,271.289,-66.548,-177.015,7.326,148.512
C03119=1186.232,271.041,-66.520,-177.018,7.324,148.513
C03120=1186.237,270.792,-66.491,-177.020,7.322,148.513
C03121=1186.241,270.544,-66.463,-177.023,7.319,148.513
C03122=1186.246,270.296,-66.435,-177.026,7.316,148.513
C03123=1186.250,270.047,-66.407,-177.028,7.314,148.513
C03124=1186.254,269.799,-66.379,-177.031,7.311,148.513
C03125=1186.259,269.550,-66.350,-177.033,7.308,148.513
C03126=1186.263,269.302,-66.322,-177.036,7.306,148.513
C03127=1186.267,269.053,-66.295,-177.039,7.303,148.513
C03128=1186.272,268.805,-66.267,-177.041,7.301,148.513
C03129=1186.277,268.557,-66.239,-177.044,7.298,148.513
C03130=1186.280,268.309,-66.211,-177.046,7.295,148.513
C03131=1186.285,268.060,-66.182,-177.049,7.293,148.514
C03132=1186.289,267.811,-66.155,-177.052,7.290,148.514
C03133=1186.294,267.563,-66.127,-177.054,7.288,148.514
C03134=1186.298,267.315,-66.099,-177.057,7.285,148.514
C03135=1186.303,267.067,-66.071,-177.059,7.282,148.514
C03136=1186.307,266.819,-66.043,-177.061,7.279,148.514
C03137=1186.311,266.569,-66.015,-177.065,7.277,148.514
C03138=1186.315,266.322,-65.988,-177.067,7.275,148.514
C03139=1186.320,266.073,-65.959,-177.070,7.272,148.514
C03140=1186.325,265.824,-65.932,-177.072,7.269,148.514
C03141=1186.329,265.576,-65.904,-177.074,7.266,148.515
C03142=1186.333,265.328,-65.876,-177.078,7.264,148.515
C03143=1186.338,265.079,-65.848,-177.080,7.262,148.515
C03144=1186.342,264.831,-65.821,-177.082,7.259,148.515
C03145=1186.346,264.583,-65.792,-177.085,7.256,148.515
C03146=1186.351,264.334,-65.765,-177.087,7.254,148.515
C03147=1186.355,264.085,-65.737,-177.091,7.251,148.515
C03148=1186.359,263.837,-65.710,-177.093,7.249,148.515
C03149=1186.364,263.589,-65.682,-177.095,7.246,148.515
C03150=1186.368,263.340,-65.654,-177.098,7.243,148.516
C03151=1186.373,263.092,-65.627,-177.101,7.241,148.516
C03152=1186.378,262.819,-65.596,-177.104,7.238,148.516
C03153=1186.383,262.546,-65.566,-177.106,7.235,148.516
C03154=1186.387,262.273,-65.536,-177.109,7.232,148.516
C03155=1186.392,262.000,-65.505,-177.112,7.229,148.516
C03156=1186.396,261.752,-65.477,-177.114,7.227,148.516
C03157=1186.401,261.504,-65.450,-177.117,7.224,148.516
C03158=1186.405,261.255,-65.422,-177.120,7.221,148.517
C03159=1186.409,261.007,-65.395,-177.122,7.219,148.517
C03160=1186.414,260.758,-65.368,-177.125,7.216,148.517
C03161=1186.418,260.510,-65.340,-177.127,7.214,148.517
C03162=1186.423,260.261,-65.312,-177.131,7.211,148.517
C03163=1186.427,260.013,-65.284,-177.133,7.209,148.517
C03164=1186.432,259.764,-65.257,-177.135,7.206,148.517
C03165=1186.436,259.515,-65.230,-177.138,7.203,148.517
C03166=1186.440,259.267,-65.202,-177.141,7.202,148.518
C03167=1186.445,259.019,-65.175,-177.144,7.199,148.518
C03168=1186.449,258.770,-65.147,-177.146,7.196,148.518
C03169=1186.454,258.522,-65.120,-177.149,7.194,148.518
C03170=1186.458,258.273,-65.093,-177.151,7.192,148.518
C03171=1186.463,258.025,-65.066,-177.154,7.189,148.518
C03172=1186.467,257.777,-65.038,-177.156,7.186,148.518
C03173=1186.471,257.528,-65.011,-177.159,7.184,148.519
C03174=1186.475,257.279,-64.984,-177.161,7.182,148.519
C03175=1186.480,257.032,-64.956,-177.164,7.179,148.519
C03176=1186.484,256.783,-64.929,-177.167,7.176,148.519
C03177=1186.488,256.534,-64.902,-177.169,7.174,148.519
C03178=1186.493,256.285,-64.875,-177.172,7.171,148.519
C03179=1186.498,256.037,-64.848,-177.174,7.169,148.519
C03180=1186.502,255.789,-64.820,-177.177,7.166,148.519
C03181=1186.507,255.541,-64.793,-177.180,7.164,148.520
C03182=1186.511,255.292,-64.766,-177.182,7.161,148.520
C03183=1186.515,255.043,-64.738,-177.185,7.159,148.520
C03184=1186.519,254.795,-64.712,-177.188,7.156,148.520
C03185=1186.524,254.546,-64.685,-177.190,7.154,148.520
C03186=1186.528,254.298,-64.657,-177.193,7.151,148.520
C03187=1186.533,254.050,-64.630,-177.195,7.149,148.520
C03188=1186.538,253.801,-64.603,-177.198,7.146,148.520
C03189=1186.542,253.552,-64.576,-177.200,7.144,148.521
C03190=1186.546,253.304,-64.549,-177.203,7.141,148.521
C03191=1186.550,253.055,-64.522,-177.206,7.139,148.521
C03192=1186.555,252.807,-64.495,-177.208,7.136,148.521
C03193=1186.559,252.558,-64.468,-177.211,7.134,148.521
C03194=1186.564,252.310,-64.441,-177.214,7.131,148.521
C03195=1186.568,252.062,-64.414,-177.216,7.129,148.521
C03196=1186.572,251.813,-64.387,-177.219,7.127,148.522
C03197=1186.577,251.564,-64.360,-177.221,7.124,148.522
C03198=1186.581,251.316,-64.333,-177.224,7.121,148.522
C03199=1186.586,251.067,-64.306,-177.227,7.120,148.522
C03200=1186.590,250.819,-64.279,-177.229,7.117,148.522
C03201=1186.595,250.570,-64.252,-177.231,7.114,148.522
C03202=1186.599,250.322,-64.225,-177.235,7.112,148.523
C03203=1186.603,250.074,-64.199,-177.237,7.110,148.523
C03204=1186.608,249.825,-64.172,-177.240,7.107,148.523
C03205=1186.613,249.577,-64.145,-177.242,7.105,148.523
C03206=1186.617,249.328,-64.118,-177.245,7.102,148.523
C03207=1186.621,249.079,-64.092,-177.248,7.100,148.523
C03208=1186.626,248.831,-64.065,-177.250,7.097,148.524
C03209=1186.630,248.582,-64.037,-177.252,7.095,148.524
C03210=1186.634,248.334,-64.011,-177.256,7.092,148.524
C03211=1186.639,248.085,-63.984,-177.258,7.090,148.524
C03212=1186.644,247.836,-63.957,-177.261,7.087,148.524
C03213=1186.648,247.588,-63.931,-177.263,7.085,148.524
C03214=1186.652,247.339,-63.904,-177.266,7.082,148.524
C03215=1186.656,247.091,-63.877,-177.269,7.080,148.525
C03216=1186.661,246.843,-63.850,-177.271,7.077,148.525
C03217=1186.666,246.593,-63.824,-177.273,7.075,148.525
C03218=1186.670,246.345,-63.798,-177.276,7.073,148.525
C03219=1186.674,246.097,-63.771,-177.279,7.070,148.525
C03220=1186.679,245.848,-63.745,-177.281,7.069,148.526
C03221=1186.683,245.599,-63.718,-177.284,7.066,148.526
C03222=1186.687,245.351,-63.691,-177.286,7.063,148.526
C03223=1186.692,245.103,-63.664,-177.290,7.061,148.526
C03224=1186.697,244.854,-63.638,-177.292,7.059,148.526
C03225=1186.701,244.606,-63.611,-177.295,7.056,148.526
C03226=1186.706,244.356,-63.585,-177.297,7.054,148.527
C03227=1186.710,244.108,-63.559,-177.300,7.051,148.527
C03228=1186.714,243.860,-63.531,-177.302,7.049,148.527
C03229=1186.719,243.612,-63.506,-177.305,7.047,148.527
C03230=1186.724,243.363,-63.479,-177.308,7.044,148.527
C03231=1186.728,243.114,-63.453,-177.310,7.042,148.527
C03232=1186.733,242.866,-63.426,-177.313,7.039,148.528
C03233=1186.737,242.618,-63.400,-177.315,7.037,148.528
C03234=1186.741,242.369,-63.373,-177.318,7.034,148.528
C03235=1186.745,242.120,-63.347,-177.321,7.033,148.528
C03236=1186.750,241.871,-63.321,-177.323,7.030,148.528
C03237=1186.754,241.623,-63.294,-177.326,7.028,148.529
C03238=1186.758,241.374,-63.268,-177.328,7.026,148.529
C03239=1186.763,241.126,-63.241,-177.332,7.023,148.529
C03240=1186.767,240.877,-63.216,-177.334,7.021,148.529
C03241=1186.773,240.629,-63.189,-177.337,7.018,148.529
C03242=1186.777,240.380,-63.163,-177.339,7.016,148.529
C03243=1186.781,240.132,-63.137,-177.341,7.014,148.529
C03244=1186.786,239.883,-63.110,-177.344,7.011,148.530
C03245=1186.790,239.634,-63.085,-177.347,7.009,148.530
C03246=1186.795,239.386,-63.058,-177.350,7.006,148.530
C03247=1186.799,239.137,-63.032,-177.352,7.004,148.530
C03248=1186.803,238.888,-63.006,-177.355,7.002,148.531
C03249=1186.808,238.640,-62.979,-177.357,6.999,148.531
C03250=1186.813,238.392,-62.954,-177.360,6.998,148.531
C03251=1186.817,238.143,-62.928,-177.363,6.995,148.531
C03252=1186.821,237.894,-62.901,-177.365,6.993,148.531
C03253=1186.826,237.645,-62.875,-177.368,6.990,148.531
C03254=1186.830,237.397,-62.849,-177.371,6.988,148.532
C03255=1186.835,237.149,-62.823,-177.373,6.986,148.532
C03256=1186.840,236.877,-62.795,-177.376,6.983,148.532
C03257=1186.844,236.606,-62.766,-177.379,6.980,148.532
C03258=1186.849,236.334,-62.738,-177.382,6.978,148.532
C03259=1186.854,236.062,-62.709,-177.385,6.976,148.533
C03260=1186.859,235.814,-62.683,-177.387,6.973,148.533
C03261=1186.863,235.565,-62.657,-177.390,6.971,148.533
C03262=1186.867,235.316,-62.631,-177.392,6.969,148.533
C03263=1186.872,235.067,-62.605,-177.395,6.966,148.534
C03264=1186.877,234.819,-62.580,-177.398,6.964,148.534
C03265=1186.881,234.571,-62.553,-177.401,6.961,148.534
C03266=1186.885,234.322,-62.528,-177.403,6.959,148.534
C03267=1186.889,234.073,-62.502,-177.406,6.957,148.534
C03268=1186.894,233.824,-62.475,-177.408,6.954,148.534
C03269=1186.899,233.576,-62.450,-177.411,6.953,148.535
C03270=1186.903,233.327,-62.424,-177.413,6.950,148.535
C03271=1186.908,233.079,-62.399,-177.416,6.948,148.535
C03272=1186.913,232.830,-62.373,-177.419,6.946,148.535
C03273=1186.917,232.581,-62.347,-177.421,6.944,148.536
C03274=1186.922,232.333,-62.321,-177.424,6.941,148.536
C03275=1186.926,232.084,-62.295,-177.427,6.939,148.536
C03276=1186.931,231.836,-62.270,-177.430,6.936,148.536
C03277=1186.935,231.587,-62.243,-177.432,6.934,148.536
C03278=1186.939,231.339,-62.218,-177.435,6.932,148.537
C03279=1186.943,231.090,-62.192,-177.437,6.929,148.537
C03280=1186.948,230.841,-62.167,-177.440,6.928,148.537
C03281=1186.952,230.592,-62.142,-177.442,6.925,148.537
C03282=1186.957,230.343,-62.115,-177.445,6.923,148.538
C03283=1186.962,230.095,-62.090,-177.448,6.921,148.538
C03284=1186.967,229.846,-62.064,-177.450,6.919,148.538
C03285=1186.971,229.598,-62.038,-177.453,6.916,148.538
C03286=1186.976,229.349,-62.013,-177.456,6.914,148.538
C03287=1186.980,229.101,-61.987,-177.458,6.912,148.539
C03288=1186.984,228.852,-61.961,-177.461,6.909,148.539
C03289=1186.989,228.604,-61.936,-177.464,6.907,148.539
C03290=1186.993,228.355,-61.910,-177.466,6.905,148.539
C03291=1186.998,228.105,-61.885,-177.469,6.903,148.540
C03292=1187.002,227.857,-61.860,-177.472,6.901,148.540
C03293=1187.007,227.609,-61.834,-177.474,6.899,148.540
C03294=1187.011,227.360,-61.808,-177.477,6.896,148.540
C03295=1187.016,227.112,-61.783,-177.479,6.894,148.540
C03296=1187.020,226.863,-61.757,-177.482,6.892,148.541
C03297=1187.025,226.614,-61.733,-177.485,6.889,148.541
C03298=1187.029,226.365,-61.707,-177.487,6.887,148.541
C03299=1187.033,226.117,-61.681,-177.490,6.885,148.541
C03300=1187.038,225.868,-61.656,-177.493,6.882,148.541
C03301=1187.043,225.619,-61.631,-177.495,6.881,148.542
C03302=1187.048,225.371,-61.605,-177.498,6.879,148.542
C03303=1187.052,225.122,-61.580,-177.501,6.876,148.542
C03304=1187.056,224.873,-61.555,-177.503,6.874,148.543
C03305=1187.061,224.625,-61.530,-177.506,6.872,148.543
C03306=1187.065,224.376,-61.504,-177.509,6.869,148.543
C03307=1187.070,224.127,-61.479,-177.511,6.867,148.543
C03308=1187.074,223.879,-61.454,-177.514,6.865,148.543
C03309=1187.079,223.630,-61.428,-177.517,6.863,148.544
C03310=1187.083,223.381,-61.403,-177.519,6.861,148.544
C03311=1187.088,223.132,-61.377,-177.522,6.859,148.544
C03312=1187.092,222.884,-61.353,-177.525,6.856,148.544
C03313=1187.096,222.635,-61.328,-177.527,6.854,148.545
C03314=1187.101,222.387,-61.302,-177.530,6.852,148.545
C03315=1187.106,222.137,-61.277,-177.532,6.850,148.545
C03316=1187.110,221.889,-61.252,-177.535,6.847,148.545
C03317=1187.115,221.640,-61.227,-177.538,6.846,148.546
C03318=1187.119,221.392,-61.202,-177.540,6.844,148.546
C03319=1187.124,221.143,-61.177,-177.543,6.841,148.546
C03320=1187.128,220.895,-61.151,-177.546,6.839,148.546
C03321=1187.133,220.645,-61.126,-177.548,6.837,148.546
C03322=1187.137,220.397,-61.102,-177.551,6.835,148.547
C03323=1187.142,220.148,-61.077,-177.554,6.832,148.547
C03324=1187.146,219.900,-61.051,-177.556,6.830,148.547
C03325=1187.151,219.650,-61.026,-177.559,6.828,148.548
C03326=1187.155,219.403,-61.001,-177.562,6.826,148.548
C03327=1187.160,219.153,-60.976,-177.564,6.824,148.548
C03328=1187.164,218.905,-60.951,-177.567,6.822,148.548
C03329=1187.169,218.656,-60.926,-177.569,6.820,148.549
C03330=1187.173,218.407,-60.902,-177.572,6.817,148.549
C03331=1187.178,218.158,-60.876,-177.575,6.815,148.549
C03332=1187.183,217.910,-60.851,-177.577,6.813,148.549
C03333=1187.187,217.662,-60.827,-177.580,6.810,148.549
C03334=1187.191,217.413,-60.802,-177.583,6.809,148.550
C03335=1187.196,217.164,-60.777,-177.585,6.807,148.550
C03336=1187.200,216.915,-60.752,-177.588,6.805,148.550
C03337=1187.205,216.667,-60.727,-177.591,6.802,148.551
C03338=1187.210,216.417,-60.702,-177.593,6.800,148.551
C03339=1187.214,216.169,-60.678,-177.596,6.798,148.551
C03340=1187.219,215.921,-60.653,-177.598,6.796,148.551
C03341=1187.223,215.671,-60.628,-177.602,6.794,148.552
C03342=1187.228,215.423,-60.604,-177.604,6.792,148.552
C03343=1187.232,215.173,-60.578,-177.606,6.790,148.552
C03344=1187.236,214.926,-60.554,-177.609,6.788,148.552
C03345=1187.241,214.677,-60.529,-177.612,6.785,148.553
C03346=1187.246,214.427,-60.504,-177.614,6.783,148.553
C03347=1187.250,214.179,-60.480,-177.617,6.781,148.553
C03348=1187.255,213.930,-60.455,-177.620,6.779,148.554
C03349=1187.259,213.682,-60.430,-177.623,6.777,148.554
C03350=1187.264,213.433,-60.405,-177.625,6.775,148.554
C03351=1187.268,213.184,-60.381,-177.628,6.773,148.554
C03352=1187.273,212.935,-60.356,-177.630,6.771,148.555
C03353=1187.277,212.687,-60.332,-177.633,6.768,148.555
C03354=1187.282,212.437,-60.307,-177.636,6.766,148.555
C03355=1187.286,212.189,-60.283,-177.639,6.764,148.555
C03356=1187.292,211.940,-60.258,-177.641,6.763,148.556
C03357=1187.295,211.692,-60.233,-177.644,6.760,148.556
C03358=1187.300,211.443,-60.209,-177.647,6.758,148.556
C03359=1187.305,211.195,-60.185,-177.649,6.756,148.557
C03360=1187.309,210.923,-60.158,-177.652,6.753,148.557
C03361=1187.315,210.653,-60.131,-177.655,6.751,148.557
C03362=1187.320,210.383,-60.105,-177.658,6.749,148.557
C03363=1187.325,210.113,-60.078,-177.660,6.747,148.558
C03364=1187.329,209.864,-60.054,-177.663,6.745,148.558
C03365=1187.334,209.615,-60.029,-177.666,6.742,148.558
C03366=1187.338,209.366,-60.005,-177.669,6.740,148.558
C03367=1187.343,209.117,-59.980,-177.671,6.738,148.559
C03368=1187.347,208.869,-59.956,-177.674,6.737,148.559
C03369=1187.352,208.620,-59.931,-177.677,6.735,148.559
C03370=1187.357,208.371,-59.907,-177.679,6.732,148.559
C03371=1187.361,208.122,-59.883,-177.682,6.730,148.560
C03372=1187.366,207.873,-59.859,-177.685,6.728,148.560
C03373=1187.370,207.625,-59.835,-177.687,6.726,148.560
C03374=1187.375,207.376,-59.810,-177.689,6.724,148.561
C03375=1187.379,207.127,-59.785,-177.693,6.722,148.561
C03376=1187.384,206.878,-59.761,-177.695,6.720,148.561
C03377=1187.389,206.630,-59.737,-177.698,6.718,148.562
C03378=1187.393,206.381,-59.713,-177.701,6.716,148.562
C03379=1187.398,206.132,-59.689,-177.703,6.714,148.562
C03380=1187.402,205.883,-59.664,-177.706,6.712,148.562
C03381=1187.407,205.634,-59.640,-177.709,6.710,148.563
C03382=1187.411,205.386,-59.616,-177.711,6.708,148.563
C03383=1187.416,205.137,-59.593,-177.714,6.706,148.563
C03384=1187.421,204.888,-59.568,-177.716,6.704,148.564
C03385=1187.425,204.639,-59.544,-177.719,6.701,148.564
C03386=1187.429,204.391,-59.520,-177.722,6.700,148.564
C03387=1187.435,204.141,-59.496,-177.724,6.697,148.564
C03388=1187.439,203.893,-59.472,-177.727,6.696,148.565
C03389=1187.443,203.644,-59.447,-177.730,6.694,148.565
C03390=1187.447,203.395,-59.423,-177.733,6.691,148.565
C03391=1187.452,203.146,-59.400,-177.735,6.689,148.566
C03392=1187.457,202.898,-59.375,-177.738,6.687,148.566
C03393=1187.461,202.649,-59.351,-177.740,6.685,148.566
C03394=1187.466,202.400,-59.328,-177.743,6.684,148.566
C03395=1187.470,202.152,-59.303,-177.746,6.682,148.567
C03396=1187.476,201.902,-59.279,-177.749,6.679,148.567
C03397=1187.480,201.653,-59.255,-177.751,6.677,148.567
C03398=1187.484,201.405,-59.231,-177.754,6.675,148.568
C03399=1187.489,201.156,-59.208,-177.756,6.673,148.568
C03400=1187.493,200.907,-59.184,-177.759,6.672,148.568
C03401=1187.498,200.658,-59.160,-177.762,6.670,148.569
C03402=1187.503,200.410,-59.136,-177.764,6.667,148.569
C03403=1187.508,200.161,-59.112,-177.767,6.665,148.569
C03404=1187.512,199.912,-59.088,-177.770,6.663,148.569
C03405=1187.516,199.662,-59.064,-177.772,6.661,148.570
C03406=1187.521,199.414,-59.040,-177.775,6.660,148.570
C03407=1187.525,199.165,-59.017,-177.777,6.658,148.570
C03408=1187.530,198.917,-58.993,-177.780,6.656,148.571
C03409=1187.534,198.668,-58.969,-177.783,6.653,148.571
C03410=1187.539,198.419,-58.945,-177.786,6.651,148.571
C03411=1187.544,198.170,-58.922,-177.788,6.650,148.572
C03412=1187.549,197.921,-58.897,-177.791,6.648,148.572
C03413=1187.553,197.672,-58.874,-177.793,6.646,148.572
C03414=1187.558,197.424,-58.850,-177.796,6.644,148.572
C03415=1187.562,197.175,-58.827,-177.799,6.642,148.573
C03416=1187.567,196.926,-58.803,-177.802,6.639,148.573
C03417=1187.572,196.677,-58.779,-177.805,6.638,148.573
C03418=1187.576,196.428,-58.756,-177.807,6.636,148.574
C03419=1187.581,196.180,-58.732,-177.809,6.634,148.574
C03420=1187.585,195.931,-58.708,-177.812,6.632,148.574
C03421=1187.590,195.682,-58.685,-177.815,6.630,148.575
C03422=1187.594,195.434,-58.661,-177.817,6.628,148.575
C03423=1187.599,195.185,-58.638,-177.820,6.626,148.575
C03424=1187.604,194.935,-58.614,-177.823,6.624,148.576
C03425=1187.609,194.686,-58.591,-177.825,6.622,148.576
C03426=1187.613,194.438,-58.567,-177.828,6.620,148.576
C03427=1187.618,194.189,-58.543,-177.831,6.618,148.576
C03428=1187.622,193.940,-58.520,-177.833,6.616,148.577
C03429=1187.627,193.691,-58.497,-177.836,6.614,148.577
C03430=1187.631,193.443,-58.473,-177.839,6.613,148.577
C03431=1187.636,193.194,-58.449,-177.841,6.611,148.578
C03432=1187.640,192.945,-58.427,-177.844,6.609,148.578
C03433=1187.645,192.696,-58.403,-177.847,6.606,148.578
C03434=1187.649,192.447,-58.380,-177.850,6.604,148.579
C03435=1187.654,192.198,-58.356,-177.852,6.603,148.579
C03436=1187.659,191.949,-58.332,-177.855,6.601,148.579
C03437=1187.663,191.700,-58.309,-177.858,6.599,148.580
C03438=1187.668,191.451,-58.286,-177.860,6.597,148.580
C03439=1187.673,191.202,-58.262,-177.862,6.595,148.580
C03440=1187.677,190.953,-58.239,-177.865,6.593,148.581
C03441=1187.681,190.704,-58.216,-177.868,6.591,148.581
C03442=1187.686,190.456,-58.192,-177.870,6.590,148.581
C03443=1187.690,190.207,-58.169,-177.873,6.588,148.582
C03444=1187.695,189.958,-58.145,-177.876,6.585,148.582
C03445=1187.700,189.710,-58.122,-177.879,6.583,148.582
C03446=1187.705,189.461,-58.099,-177.882,6.582,148.583
C03447=1187.709,189.212,-58.076,-177.884,6.580,148.583
C03448=1187.714,188.963,-58.053,-177.886,6.578,148.583
C03449=1187.718,188.714,-58.030,-177.889,6.576,148.583
C03450=1187.723,188.465,-58.006,-177.892,6.574,148.584
C03451=1187.728,188.216,-57.983,-177.894,6.572,148.584
C03452=1187.732,187.967,-57.960,-177.897,6.571,148.585
C03453=1187.737,187.719,-57.937,-177.900,6.569,148.585
C03454=1187.742,187.470,-57.914,-177.902,6.567,148.585
C03455=1187.747,187.221,-57.890,-177.905,6.565,148.586
C03456=1187.750,186.972,-57.868,-177.908,6.563,148.586
C03457=1187.755,186.723,-57.844,-177.910,6.561,148.586
C03458=1187.760,186.474,-57.821,-177.913,6.559,148.586
C03459=1187.765,186.224,-57.798,-177.916,6.557,148.587
C03460=1187.769,185.976,-57.776,-177.919,6.555,148.587
C03461=1187.774,185.727,-57.752,-177.921,6.553,148.587
C03462=1187.779,185.478,-57.729,-177.924,6.551,148.588
C03463=1187.783,185.229,-57.706,-177.927,6.550,148.588
C03464=1187.788,184.960,-57.681,-177.929,6.548,148.589
C03465=1187.793,184.690,-57.656,-177.932,6.546,148.589
C03466=1187.798,184.420,-57.632,-177.935,6.543,148.589
C03467=1187.803,184.151,-57.607,-177.938,6.542,148.590
C03468=1187.808,183.902,-57.583,-177.940,6.540,148.590
C03469=1187.812,183.653,-57.561,-177.943,6.538,148.590
C03470=1187.817,183.405,-57.538,-177.946,6.536,148.591
C03471=1187.822,183.155,-57.516,-177.948,6.534,148.591
C03472=1187.826,182.906,-57.492,-177.951,6.533,148.591
C03473=1187.831,182.657,-57.469,-177.954,6.531,148.592
C03474=1187.836,182.409,-57.447,-177.956,6.529,148.592
C03475=1187.841,182.159,-57.424,-177.959,6.527,148.592
C03476=1187.845,181.911,-57.401,-177.962,6.526,148.593
C03477=1187.849,181.662,-57.378,-177.964,6.524,148.593
C03478=1187.855,181.413,-57.355,-177.967,6.522,148.593
C03479=1187.859,181.164,-57.333,-177.969,6.520,148.594
C03480=1187.863,180.915,-57.309,-177.972,6.518,148.594
C03481=1187.867,180.666,-57.287,-177.975,6.516,148.594
C03482=1187.873,180.417,-57.264,-177.977,6.514,148.595
C03483=1187.877,180.169,-57.242,-177.981,6.512,148.595
C03484=1187.882,179.919,-57.219,-177.983,6.510,148.595
C03485=1187.886,179.670,-57.196,-177.986,6.508,148.596
C03486=1187.891,179.422,-57.173,-177.989,6.506,148.596
C03487=1187.896,179.173,-57.151,-177.991,6.505,148.596
C03488=1187.900,178.924,-57.128,-177.994,6.503,148.597
C03489=1187.905,178.675,-57.106,-177.997,6.501,148.597
C03490=1187.910,178.426,-57.083,-177.999,6.499,148.598
C03491=1187.914,178.177,-57.060,-178.002,6.498,148.598
C03492=1187.919,177.927,-57.037,-178.005,6.496,148.598
C03493=1187.923,177.679,-57.015,-178.007,6.494,148.599
C03494=1187.928,177.430,-56.992,-178.010,6.492,148.599
C03495=1187.932,177.181,-56.969,-178.013,6.490,148.599
C03496=1187.938,176.932,-56.947,-178.015,6.489,148.600
C03497=1187.942,176.683,-56.924,-178.018,6.487,148.600
C03498=1187.946,176.434,-56.902,-178.021,6.485,148.600
C03499=1187.952,176.185,-56.880,-178.023,6.483,148.601
C03500=1187.956,175.936,-56.857,-178.026,6.481,148.601
C03501=1187.961,175.687,-56.835,-178.029,6.480,148.602
C03502=1187.965,175.439,-56.812,-178.031,6.478,148.602
C03503=1187.970,175.189,-56.790,-178.033,6.477,148.602
C03504=1187.975,174.941,-56.767,-178.036,6.475,148.603
C03505=1187.979,174.692,-56.745,-178.039,6.473,148.603
C03506=1187.983,174.442,-56.723,-178.041,6.472,148.603
C03507=1187.989,174.194,-56.700,-178.044,6.470,148.604
C03508=1187.993,173.945,-56.678,-178.047,6.468,148.604
C03509=1187.999,173.696,-56.656,-178.049,6.466,148.604
C03510=1188.003,173.447,-56.633,-178.052,6.464,148.605
C03511=1188.007,173.198,-56.611,-178.055,6.463,148.605
C03512=1188.012,172.949,-56.589,-178.057,6.461,148.606
C03513=1188.016,172.700,-56.566,-178.060,6.459,148.606
C03514=1188.021,172.451,-56.544,-178.063,6.457,148.606
C03515=1188.026,172.202,-56.522,-178.066,6.456,148.607
C03516=1188.030,171.953,-56.499,-178.068,6.454,148.607
C03517=1188.035,171.704,-56.477,-178.071,6.452,148.607
C03518=1188.039,171.455,-56.455,-178.074,6.450,148.608
C03519=1188.045,171.206,-56.433,-178.076,6.448,148.608
C03520=1188.049,170.957,-56.410,-178.079,6.447,148.608
C03521=1188.054,170.709,-56.388,-178.082,6.445,148.609
C03522=1188.058,170.459,-56.366,-178.084,6.443,148.609
C03523=1188.064,170.210,-56.344,-178.087,6.441,148.610
C03524=1188.068,169.961,-56.322,-178.090,6.439,148.610
C03525=1188.073,169.712,-56.300,-178.092,6.438,148.610
C03526=1188.077,169.464,-56.278,-178.095,6.436,148.611
C03527=1188.082,169.215,-56.255,-178.098,6.434,148.611
C03528=1188.087,168.965,-56.233,-178.100,6.432,148.611
C03529=1188.092,168.717,-56.212,-178.102,6.431,148.612
C03530=1188.096,168.467,-56.190,-178.105,6.430,148.612
C03531=1188.101,168.219,-56.168,-178.108,6.428,148.612
C03532=1188.105,167.969,-56.146,-178.110,6.426,148.613
C03533=1188.111,167.721,-56.124,-178.113,6.424,148.613
C03534=1188.114,167.472,-56.101,-178.116,6.422,148.614
C03535=1188.119,167.223,-56.079,-178.118,6.421,148.614
C03536=1188.124,166.974,-56.057,-178.121,6.419,148.614
C03537=1188.128,166.725,-56.035,-178.124,6.417,148.615
C03538=1188.133,166.476,-56.013,-178.126,6.415,148.615
C03539=1188.138,166.227,-55.992,-178.129,6.414,148.615
C03540=1188.143,165.978,-55.969,-178.132,6.412,148.616
C03541=1188.148,165.729,-55.947,-178.135,6.410,148.616
C03542=1188.152,165.480,-55.925,-178.137,6.408,148.617
C03543=1188.157,165.231,-55.904,-178.140,6.408,148.617
C03544=1188.161,164.982,-55.882,-178.142,6.406,148.618
C03545=1188.166,164.733,-55.860,-178.145,6.404,148.618
C03546=1188.170,164.484,-55.838,-178.148,6.402,148.618
C03547=1188.175,164.234,-55.817,-178.150,6.400,148.619
C03548=1188.180,163.986,-55.795,-178.153,6.399,148.619
C03549=1188.184,163.736,-55.773,-178.156,6.397,148.619
C03550=1188.189,163.488,-55.751,-178.159,6.395,148.620
C03551=1188.193,163.238,-55.729,-178.161,6.393,148.620
C03552=1188.198,162.990,-55.708,-178.164,6.392,148.620
C03553=1188.203,162.741,-55.686,-178.166,6.391,148.621
C03554=1188.208,162.492,-55.664,-178.169,6.389,148.621
C03555=1188.212,162.243,-55.642,-178.171,6.387,148.622
C03556=1188.217,161.993,-55.621,-178.174,6.385,148.622
C03557=1188.222,161.745,-55.599,-178.177,6.384,148.622
C03558=1188.227,161.496,-55.578,-178.180,6.382,148.623
C03559=1188.231,161.247,-55.556,-178.183,6.380,148.623
C03560=1188.236,160.998,-55.534,-178.185,6.379,148.624
C03561=1188.241,160.749,-55.513,-178.188,6.377,148.624
C03562=1188.245,160.499,-55.491,-178.190,6.376,148.624
C03563=1188.250,160.251,-55.469,-178.193,6.374,148.625
C03564=1188.254,160.001,-55.447,-178.195,6.372,148.625
C03565=1188.260,159.752,-55.426,-178.198,6.370,148.626
C03566=1188.264,159.503,-55.404,-178.201,6.369,148.626
C03567=1188.269,159.254,-55.382,-178.203,6.367,148.626
C03568=1188.273,158.985,-55.360,-178.207,6.365,148.627
C03569=1188.280,158.716,-55.337,-178.209,6.364,148.627
C03570=1188.284,158.448,-55.313,-178.212,6.362,148.628
C03571=1188.289,158.179,-55.290,-178.215,6.360,148.628
C03572=1188.294,157.929,-55.268,-178.218,6.359,148.629
C03573=1188.299,157.680,-55.247,-178.220,6.357,148.629
C03574=1188.303,157.432,-55.226,-178.223,6.355,148.629
C03575=1188.307,157.182,-55.204,-178.226,6.353,148.630
C03576=1188.312,156.933,-55.183,-178.229,6.352,148.630
C03577=1188.317,156.684,-55.161,-178.231,6.351,148.630
C03578=1188.323,156.435,-55.140,-178.233,6.349,148.631
C03579=1188.327,156.186,-55.118,-178.236,6.347,148.631
C03580=1188.332,155.937,-55.096,-178.239,6.345,148.632
C03581=1188.336,155.688,-55.076,-178.242,6.344,148.632
C03582=1188.341,155.440,-55.054,-178.245,6.342,148.633
C03583=1188.346,155.190,-55.033,-178.247,6.340,148.633
C03584=1188.350,154.941,-55.011,-178.249,6.339,148.633
C03585=1188.356,154.692,-54.990,-178.252,6.338,148.634
C03586=1188.359,154.443,-54.969,-178.255,6.336,148.634
C03587=1188.364,154.193,-54.948,-178.257,6.334,148.634
C03588=1188.369,153.945,-54.926,-178.260,6.332,148.635
C03589=1188.374,153.696,-54.905,-178.263,6.331,148.635
C03590=1188.378,153.447,-54.884,-178.265,6.330,148.636
C03591=1188.383,153.197,-54.863,-178.268,6.328,148.636
C03592=1188.388,152.949,-54.841,-178.271,6.326,148.637
C03593=1188.393,152.699,-54.820,-178.273,6.325,148.637
C03594=1188.398,152.450,-54.800,-178.276,6.323,148.637
C03595=1188.402,152.202,-54.778,-178.279,6.321,148.638
C03596=1188.407,151.952,-54.757,-178.281,6.320,148.638
C03597=1188.411,151.703,-54.736,-178.284,6.319,148.639
C03598=1188.416,151.454,-54.715,-178.287,6.317,148.639
C03599=1188.421,151.205,-54.694,-178.289,6.315,148.639
C03600=1188.426,150.956,-54.672,-178.292,6.313,148.640
C03601=1188.430,150.707,-54.651,-178.295,6.312,148.640
C03602=1188.435,150.457,-54.630,-178.297,6.311,148.641
C03603=1188.440,150.209,-54.609,-178.300,6.309,148.641
C03604=1188.445,149.960,-54.588,-178.303,6.307,148.642
C03605=1188.450,149.711,-54.567,-178.305,6.306,148.642
C03606=1188.454,149.462,-54.546,-178.308,6.304,148.642
C03607=1188.459,149.212,-54.525,-178.310,6.303,148.643
C03608=1188.464,148.963,-54.504,-178.313,6.301,148.643
C03609=1188.468,148.715,-54.483,-178.316,6.300,148.644
C03610=1188.473,148.465,-54.462,-178.319,6.298,148.644
C03611=1188.477,148.216,-54.442,-178.321,6.296,148.645
C03612=1188.483,147.967,-54.421,-178.324,6.295,148.645
C03613=1188.487,147.719,-54.399,-178.326,6.294,148.645
C03614=1188.491,147.469,-54.378,-178.329,6.292,148.646
C03615=1188.496,147.220,-54.357,-178.332,6.290,148.646
C03616=1188.501,146.971,-54.337,-178.335,6.289,148.647
C03617=1188.506,146.721,-54.316,-178.337,6.288,148.647
C03618=1188.511,146.472,-54.295,-178.340,6.286,148.647
C03619=1188.515,146.224,-54.274,-178.342,6.284,148.648
C03620=1188.521,145.975,-54.253,-178.345,6.282,148.648
C03621=1188.525,145.726,-54.232,-178.348,6.282,148.649
C03622=1188.530,145.476,-54.211,-178.350,6.280,148.649
C03623=1188.535,145.227,-54.191,-178.353,6.278,148.650
C03624=1188.540,144.978,-54.170,-178.356,6.276,148.650
C03625=1188.544,144.728,-54.149,-178.358,6.275,148.650
C03626=1188.549,144.479,-54.128,-178.361,6.274,148.651
C03627=1188.553,144.231,-54.107,-178.364,6.272,148.651
C03628=1188.558,143.982,-54.086,-178.366,6.271,148.652
C03629=1188.563,143.733,-54.066,-178.369,6.269,148.652
C03630=1188.567,143.484,-54.046,-178.371,6.268,148.653
C03631=1188.572,143.235,-54.025,-178.374,6.266,148.653
C03632=1188.577,142.986,-54.004,-178.377,6.265,148.654
C03633=1188.582,142.736,-53.983,-178.380,6.263,148.654
C03634=1188.586,142.487,-53.963,-178.382,6.261,148.654
C03635=1188.591,142.238,-53.942,-178.384,6.260,148.655
C03636=1188.596,141.989,-53.922,-178.388,6.259,148.655
C03637=1188.600,141.740,-53.901,-178.390,6.257,148.656
C03638=1188.605,141.491,-53.880,-178.393,6.255,148.656
C03639=1188.610,141.242,-53.860,-178.395,6.254,148.656
C03640=1188.615,140.993,-53.839,-178.398,6.253,148.657
C03641=1188.619,140.744,-53.819,-178.401,6.251,148.657
C03642=1188.624,140.495,-53.798,-178.404,6.249,148.658
C03643=1188.629,140.245,-53.778,-178.406,6.248,148.658
C03644=1188.634,139.996,-53.758,-178.408,6.247,148.659
C03645=1188.638,139.747,-53.737,-178.411,6.245,148.659
C03646=1188.643,139.498,-53.716,-178.414,6.243,148.660
